(* CODESYS project machinemanage.library
   Title: MachineManage
   Version: 1.3.0.0
   Placeholder: MachineManage
   Company: Secote

Project tree, tasks and I/O mapping:
  libraries: Recipe Management, * (System); Tc2_DataExchange, * (Beckhoff Automation GmbH); Tc2_MC2, * (Beckhoff Automation GmbH); Tc2_MC2_Camming, * (Beckhoff Automation GmbH); Tc2_ModbusSrv, * (Beckhoff Automation GmbH); Tc2_Standard, * (Beckhoff Automation GmbH); Tc2_System, * (Beckhoff Automation GmbH); Tc2_TcpIp, * (Beckhoff Automation GmbH); Tc2_Utilities, * (Beckhoff Automation GmbH); Tc3_IotBase, * (Beckhoff Automation GmbH); Tc3_JsonXml, * (Beckhoff Automation GmbH); Tc3_MC2_AdvancedHoming, * (Beckhoff Automation GmbH); Tc3_PLCopen_OpcUa, * (Beckhoff Automation GmbH); VisuDialogs, * (System)
  Axis/
    DUTs/
      data type ST_Axis
      data type ST_AxisControl
      data type ST_AxisControlHome
      data type ST_AxisControlJog
      data type ST_AxisControlMove
      data type ST_AxisData
      data type ST_AxisInfo
      data type ST_AxisInput
      data type ST_AxisLock
      data type ST_AxisMode
      data type ST_AxisStatus
      data type ST_AxisTorque
    POUs/
      function block FB_Axis [ST]: A_ControlRest, A_Error, A_Home, A_Init, A_Jog, A_Memory, A_MoveAbsolute, A_MoveRelative, A_Power, A_Rest, A_Stop, A_Teach, M_GetAbsDone, M_GetRelDone, M_Home, M_Jog, M_MoveAbs, M_MoveRel
    VISUs/
      visualisation CtrlAxis
      visualisation CtrlAxisGroup
      text list TextHomeMode
  AxisCam/
    function block FB_AxisCam [ST]: A_Run, M_Semicircle
  Convert/
    function Data_TO_Data [ST]
  CycleTime/
    function block FB_CycleTime [ST]
    function block FB_CycleTime1 [ST]
  Cylinder/
    DUTs/
      data type ST_Cylinder
      data type ST_CylinderControl
      data type ST_CylinderData
      data type ST_CylinderInfo
      data type ST_CylinderInput
      data type ST_CylinderLock
      data type ST_CylinderOutput
      data type ST_CylinderStatus
    POUs/
      function block FB_Cylinder [ST]: A_ControlRest, A_Error, A_Home, A_Init, A_Memory, A_Off, A_Work, M_HomeRequest, M_OffRequest, M_WorkRequest
    VISUs/
      visualisation CtrlCylinder
      visualisation CtrlCylinderGroup
  Error/
    DUTs/
      data type E_ErrorCategory
      data type ST_Error
      data type ST_ErrorGroup
      data type ST_ErrorInfo
    POUs/
      function block FB_ErrorTag [ST]
      function block FB_ErrorTagStation [ST]
      function M_GetCategory [ST]
    VISUs/
      visualisation CtrlError
      visualisation CtrlError1
      visualisation CtrlErrorGroup
  File/
    DUTs/
      data type E_Directory
      data type ST_FileHandle
      data type ST_FileHandleData
      data type ST_FileHandleRead
      data type ST_FileHandleStatus
      data type ST_FilHandleControl
    POUs/
      function block FB_DirectoryHelper [ST]: A_Run
      function block FB_DirectoryHelper1 [ST]
      function block FB_FileHandle [ST]: A_Error, A_Read, A_Rest, A_Run, A_Status, A_Write
      function block FB_FileHelper [ST]
      function block FB_LogHelper [ST]: A_Run, A_Status
      function block FB_LogHelper_B [ST]: A_AddTail
      function block FB_LogHelper_E [ST]: A_Run, A_Status
      function block FB_LogHelper_E_B [ST]: A_AddTail
      function block FB_LogHelper1 [ST]: M_AddTail
  Hive/
    DUTs/
      data type E_HiveState
      data type ST_Hive
      data type ST_HiveAddress
      data type ST_HiveControl
      data type ST_HiveData
      data type ST_HiveInfo
      data type ST_HiveMachineData
    POUs/
      function block FB_Hive [ST]: A_Data, A_Init, A_Mode, A_State, A_Ton, M_Data, M_DateTime, M_Join0, M_ModeOff, M_ModeOn, M_State
      program P_Hive [ST]: M_Data, M_Error, M_GetData, M_Mode, M_State
  Http/
    DOTs/
      data type E_HttpRequestOrder
      data type ST_HttpClient
      data type ST_HttpClientControl
      data type ST_HttpClientData
      data type ST_HttpClientInfo
      data type ST_HttpClientStatus
    POUs/
      function block FB_HttpClient [ST]: A_Error, A_Init, A_Run, SendRequest
      function block FB_HttpClient1 [ST]: A_Run, SendRequest
    VISUs/
  ImagePool/
    Image/
      AlarmActive.png
      AlarmInactive.png
      AlarmInactive_gray.png
      auto_mode_80x80.png
      axis.png
      axis_black_80x80.png
      axis_gray_80x80.png
      axis_red_80x80.png
      background.png
      btn_off_switch.png
      btn_off_switch_silde.png
      btn_on_switch.png
      btn_on_switch_silde.png
      BtnData1.png
      BtnData2.png
      BtnFile1.png
      BtnFile2.png
      BtnHalt1.png
      BtnHalt2.png
      BtnHome1.png
      BtnHome2.png
      BtnInfo1.png
      BtnInfo2.png
      BtnLogin1.png
      BtnLogin2.png
      BtnOFF.png
      BtnON.png
      BtnPause1.png
      BtnPause2.png
      BtnSave1.png
      BtnSave2.png
      BtnSetting1.png
      BtnSetting2.png
      BtnStart1.png
      BtnStart2.png
      BtnVision1.png
      BtnVision2.png
      BtnVision3.png
      BtnVision4.png
      Button1.png
      Button10.png
      Button11.png
      Button13.png
      Button14.png
      Button15.png
      Button16.png
      Button17.png
      Button2.png
      Button3.png
      Button4.png
      Button5.png
      Button6.png
      Button7.png
      Button8.png
      Button9.png
      buzzer1.png
      buzzer2.png
      chinese.png
      cross-512.png
      Cylinder1.png
      English.png
      File.png
      Hindi.png
      ico_actuator_black.png
      ico_actuator_gray.png
      ico_actuator_red.png
      ico_analytic.png
      ico_analytic_100x100.png
      ico_analytic_off_100x100.png
      ico_apply.png
      ico_barcodeScanner.png
      ico_barcodeScanner_black.png
      ico_barcodeScanner_gray.png
      ico_barcodeScanner_red.png
      ico_calibrate.png
      ico_calibrate2.png
      ico_calibrate2_80x80.png
      ico_chart_bar.png
      ico_chart_half_pie.png
      ico_chart_line.png
      ico_chart_pie.png
      ico_clock_black.png
      ico_close.png
      ico_close_win.png
      ico_conveyor_big.png
      ico_conveyor_black.png
      ico_conveyor_gray.png
      ico_conveyor_red.png
      ico_diskdrive.png
      ico_folder.png
      ico_folder_.png
      ico_force_black_400X400.png
      ico_force_black_80X80.png
      ico_force_gray_80X80.png
      ico_force_red_80X80.png
      ico_HMI.png
      ico_info.png
      ico_io_300x300.png
      ico_max_win.png
      ico_menu_alarm.png
      ico_menu_backward.png
      ico_menu_camFolder.png
      ico_menu_clean.png
      ico_menu_excel.png
      ico_menu_forward.png
      ico_menu_home.png
      ico_menu_info.png
      ico_menu_options.png
      ico_menu_options_big.png
      ico_menu_pause.png
      ico_menu_play.png
      ico_menu_save.png
      ico_menu_stat.png
      ico_menu_step.png
      ico_menu_stop.png
      ico_menu_stop_black.png
      ico_menu_user.png
      ico_menu_user_logged_in.png
      ico_menu_vision.png
      ico_min_win.png
      ico_next.png
      ico_pneumatic_actuator.png
      ico_prev.png
      ico_robot_big.png
      ico_robot_black.png
      ico_robot_gray.png
      ico_robot_red.png
      ico_service.png
      ico_small_light_000.png
      ico_small_light_001.png
      ico_small_light_010.png
      ico_small_light_011.png
      ico_small_light_100.png
      ico_small_light_101.png
      ico_small_light_110.png
      ico_small_light_111.png
      ico_small_light_GGG.png
      ico_small_light_gray.png
      ico_small_light_green.png
      ico_small_light_red.png
      ico_stopper.png
      ico_tray.png
      ico_tray_black.png
      ico_tray_gray.png
      ico_tray_red.png
      ico_upload.png
      ico_usb.png
      ico_usb_small.png
      ico_vacuum_256x256.ico
      ico_vacuum_black_50x50.png
      ico_vacuum_cleaner_512x512.png
      ico_vacuum_cleaner_black_80x80.png
      ico_vacuum_cleaner_gray_80x80.png
      ico_vacuum_cleaner_red_80x80.png
      ico_vacuum_gray_50x50.png
      ico_vacuum_red_50x50.png
      ico_vacuumgauge_1200x1200.png
      ico_vacuumgauge_64x64.png
      ico_vacuumgauge_black_80x80.png
      ico_vacuumgauge_gray_80x80.png
      ico_vacuumgauge_red_80x80.png
      ico_version_history.png
      ico_vision_black.png
      ico_vision_gray.png
      ico_vision_red.png
      ico_wireless.png
      ico_wireless_51x40.png
      IO1.png
      IO2.png
      lamp.png
      lightbulb-default-80x80.png
      lightbulb-full-size.png
      lightbulb-off-80x80.png
      lightbulb-on-80x80.png
      Lock.jpg
      LUX.PNG
      manual_mode_80x80.png
      nav_first.png
      nav_last.png
      next.png
      NoImage.jpg
      phone.png
      phone1.png
      Pressure.png
      prev.png
      process.png
      right_arrow_128px_1205479_easyicon.net.ico
      right_arrow_128px_1205479_easyicon.net1.ico
      saveScreenshot.png
      service.png
      Setting.png
      Setting1.png
      Time.png
      Vietnamese.png
      warning.png
      zip_logs.png
    image pool ImagePool
  00000000-0000-0000-0000-000000000000|ImagePool\Image\AlarmActive.png
  00000000-0000-0000-0000-000000000000|ImagePool\Image\AlarmInactive.png
  00000000-0000-0000-0000-000000000000|ImagePool\Image\AlarmInactive_gray.png
  00000000-0000-0000-0000-000000000000|ImagePool\Image\auto_mode_80x80.png
  00000000-0000-0000-0000-000000000000|ImagePool\Image\axis.png
  00000000-0000-0000-0000-000000000000|ImagePool\Image\axis_black_80x80.png
  00000000-0000-0000-0000-000000000000|ImagePool\Image\axis_gray_80x80.png
  00000000-0000-0000-0000-000000000000|ImagePool\Image\axis_red_80x80.png
  00000000-0000-0000-0000-000000000000|ImagePool\Image\background.png
  00000000-0000-0000-0000-000000000000|ImagePool\Image\btn_off_switch.png
  00000000-0000-0000-0000-000000000000|ImagePool\Image\btn_off_switch_silde.png
  00000000-0000-0000-0000-000000000000|ImagePool\Image\btn_on_switch.png
  00000000-0000-0000-0000-000000000000|ImagePool\Image\btn_on_switch_silde.png
  00000000-0000-0000-0000-000000000000|ImagePool\Image\BtnData1.png
  00000000-0000-0000-0000-000000000000|ImagePool\Image\BtnData2.png
  00000000-0000-0000-0000-000000000000|ImagePool\Image\BtnFile1.png
  00000000-0000-0000-0000-000000000000|ImagePool\Image\BtnFile2.png
  00000000-0000-0000-0000-000000000000|ImagePool\Image\BtnHalt1.png
  00000000-0000-0000-0000-000000000000|ImagePool\Image\BtnHalt2.png
  00000000-0000-0000-0000-000000000000|ImagePool\Image\BtnHome1.png
  00000000-0000-0000-0000-000000000000|ImagePool\Image\BtnHome2.png
  00000000-0000-0000-0000-000000000000|ImagePool\Image\BtnInfo1.png
  00000000-0000-0000-0000-000000000000|ImagePool\Image\BtnInfo2.png
  00000000-0000-0000-0000-000000000000|ImagePool\Image\BtnLogin1.png
  00000000-0000-0000-0000-000000000000|ImagePool\Image\BtnLogin2.png
  00000000-0000-0000-0000-000000000000|ImagePool\Image\BtnOFF.png
  00000000-0000-0000-0000-000000000000|ImagePool\Image\BtnON.png
  00000000-0000-0000-0000-000000000000|ImagePool\Image\BtnPause1.png
  00000000-0000-0000-0000-000000000000|ImagePool\Image\BtnPause2.png
  00000000-0000-0000-0000-000000000000|ImagePool\Image\BtnSave1.png
  00000000-0000-0000-0000-000000000000|ImagePool\Image\BtnSave2.png
  00000000-0000-0000-0000-000000000000|ImagePool\Image\BtnSetting1.png
  00000000-0000-0000-0000-000000000000|ImagePool\Image\BtnSetting2.png
  00000000-0000-0000-0000-000000000000|ImagePool\Image\BtnStart1.png
  00000000-0000-0000-0000-000000000000|ImagePool\Image\BtnStart2.png
  00000000-0000-0000-0000-000000000000|ImagePool\Image\BtnVision1.png
  00000000-0000-0000-0000-000000000000|ImagePool\Image\BtnVision2.png
  00000000-0000-0000-0000-000000000000|ImagePool\Image\BtnVision3.png
  00000000-0000-0000-0000-000000000000|ImagePool\Image\BtnVision4.png
  00000000-0000-0000-0000-000000000000|ImagePool\Image\Button1.png
  00000000-0000-0000-0000-000000000000|ImagePool\Image\Button10.png
  00000000-0000-0000-0000-000000000000|ImagePool\Image\Button11.png
  00000000-0000-0000-0000-000000000000|ImagePool\Image\Button13.png
  00000000-0000-0000-0000-000000000000|ImagePool\Image\Button14.png
  00000000-0000-0000-0000-000000000000|ImagePool\Image\Button15.png
  00000000-0000-0000-0000-000000000000|ImagePool\Image\Button16.png
  00000000-0000-0000-0000-000000000000|ImagePool\Image\Button17.png
  00000000-0000-0000-0000-000000000000|ImagePool\Image\Button2.png
  00000000-0000-0000-0000-000000000000|ImagePool\Image\Button3.png
  00000000-0000-0000-0000-000000000000|ImagePool\Image\Button4.png
  00000000-0000-0000-0000-000000000000|ImagePool\Image\Button5.png
  00000000-0000-0000-0000-000000000000|ImagePool\Image\Button6.png
  00000000-0000-0000-0000-000000000000|ImagePool\Image\Button7.png
  00000000-0000-0000-0000-000000000000|ImagePool\Image\Button8.png
  00000000-0000-0000-0000-000000000000|ImagePool\Image\Button9.png
  00000000-0000-0000-0000-000000000000|ImagePool\Image\buzzer1.png
  00000000-0000-0000-0000-000000000000|ImagePool\Image\buzzer2.png
  00000000-0000-0000-0000-000000000000|ImagePool\Image\chinese.png
  00000000-0000-0000-0000-000000000000|ImagePool\Image\cross-512.png
  00000000-0000-0000-0000-000000000000|ImagePool\Image\Cylinder1.png
  00000000-0000-0000-0000-000000000000|ImagePool\Image\English.png
  00000000-0000-0000-0000-000000000000|ImagePool\Image\File.png
  00000000-0000-0000-0000-000000000000|ImagePool\Image\Hindi.png
  00000000-0000-0000-0000-000000000000|ImagePool\Image\ico_actuator_black.png
  00000000-0000-0000-0000-000000000000|ImagePool\Image\ico_actuator_gray.png
  00000000-0000-0000-0000-000000000000|ImagePool\Image\ico_actuator_red.png
  00000000-0000-0000-0000-000000000000|ImagePool\Image\ico_analytic.png
  00000000-0000-0000-0000-000000000000|ImagePool\Image\ico_analytic_100x100.png
  00000000-0000-0000-0000-000000000000|ImagePool\Image\ico_analytic_off_100x100.png
  00000000-0000-0000-0000-000000000000|ImagePool\Image\ico_apply.png
  00000000-0000-0000-0000-000000000000|ImagePool\Image\ico_barcodeScanner.png
  00000000-0000-0000-0000-000000000000|ImagePool\Image\ico_barcodeScanner_black.png
  00000000-0000-0000-0000-000000000000|ImagePool\Image\ico_barcodeScanner_gray.png
  00000000-0000-0000-0000-000000000000|ImagePool\Image\ico_barcodeScanner_red.png
  00000000-0000-0000-0000-000000000000|ImagePool\Image\ico_calibrate.png
  00000000-0000-0000-0000-000000000000|ImagePool\Image\ico_calibrate2.png
  00000000-0000-0000-0000-000000000000|ImagePool\Image\ico_calibrate2_80x80.png
  00000000-0000-0000-0000-000000000000|ImagePool\Image\ico_chart_bar.png
  00000000-0000-0000-0000-000000000000|ImagePool\Image\ico_chart_half_pie.png
  00000000-0000-0000-0000-000000000000|ImagePool\Image\ico_chart_line.png
  00000000-0000-0000-0000-000000000000|ImagePool\Image\ico_chart_pie.png
  00000000-0000-0000-0000-000000000000|ImagePool\Image\ico_clock_black.png
  00000000-0000-0000-0000-000000000000|ImagePool\Image\ico_close.png
  00000000-0000-0000-0000-000000000000|ImagePool\Image\ico_close_win.png
  00000000-0000-0000-0000-000000000000|ImagePool\Image\ico_conveyor_big.png
  00000000-0000-0000-0000-000000000000|ImagePool\Image\ico_conveyor_black.png
  00000000-0000-0000-0000-000000000000|ImagePool\Image\ico_conveyor_gray.png
  00000000-0000-0000-0000-000000000000|ImagePool\Image\ico_conveyor_red.png
  00000000-0000-0000-0000-000000000000|ImagePool\Image\ico_diskdrive.png
  00000000-0000-0000-0000-000000000000|ImagePool\Image\ico_folder.png
  00000000-0000-0000-0000-000000000000|ImagePool\Image\ico_folder_.png
  00000000-0000-0000-0000-000000000000|ImagePool\Image\ico_force_black_400X400.png
  00000000-0000-0000-0000-000000000000|ImagePool\Image\ico_force_black_80X80.png
  00000000-0000-0000-0000-000000000000|ImagePool\Image\ico_force_gray_80X80.png
  00000000-0000-0000-0000-000000000000|ImagePool\Image\ico_force_red_80X80.png
  00000000-0000-0000-0000-000000000000|ImagePool\Image\ico_HMI.png
  00000000-0000-0000-0000-000000000000|ImagePool\Image\ico_info.png
  00000000-0000-0000-0000-000000000000|ImagePool\Image\ico_io_300x300.png
  00000000-0000-0000-0000-000000000000|ImagePool\Image\ico_max_win.png
  00000000-0000-0000-0000-000000000000|ImagePool\Image\ico_menu_alarm.png
  00000000-0000-0000-0000-000000000000|ImagePool\Image\ico_menu_backward.png
  00000000-0000-0000-0000-000000000000|ImagePool\Image\ico_menu_camFolder.png
  00000000-0000-0000-0000-000000000000|ImagePool\Image\ico_menu_clean.png
  00000000-0000-0000-0000-000000000000|ImagePool\Image\ico_menu_excel.png
  00000000-0000-0000-0000-000000000000|ImagePool\Image\ico_menu_forward.png
  00000000-0000-0000-0000-000000000000|ImagePool\Image\ico_menu_home.png
  00000000-0000-0000-0000-000000000000|ImagePool\Image\ico_menu_info.png
  00000000-0000-0000-0000-000000000000|ImagePool\Image\ico_menu_options.png
  00000000-0000-0000-0000-000000000000|ImagePool\Image\ico_menu_options_big.png
  00000000-0000-0000-0000-000000000000|ImagePool\Image\ico_menu_pause.png
  00000000-0000-0000-0000-000000000000|ImagePool\Image\ico_menu_play.png
  00000000-0000-0000-0000-000000000000|ImagePool\Image\ico_menu_save.png
  00000000-0000-0000-0000-000000000000|ImagePool\Image\ico_menu_stat.png
  00000000-0000-0000-0000-000000000000|ImagePool\Image\ico_menu_step.png
  00000000-0000-0000-0000-000000000000|ImagePool\Image\ico_menu_stop.png
  00000000-0000-0000-0000-000000000000|ImagePool\Image\ico_menu_stop_black.png
  00000000-0000-0000-0000-000000000000|ImagePool\Image\ico_menu_user.png
  00000000-0000-0000-0000-000000000000|ImagePool\Image\ico_menu_user_logged_in.png
  00000000-0000-0000-0000-000000000000|ImagePool\Image\ico_menu_vision.png
  00000000-0000-0000-0000-000000000000|ImagePool\Image\ico_min_win.png
  00000000-0000-0000-0000-000000000000|ImagePool\Image\ico_next.png
  00000000-0000-0000-0000-000000000000|ImagePool\Image\ico_pneumatic_actuator.png
  00000000-0000-0000-0000-000000000000|ImagePool\Image\ico_prev.png
  00000000-0000-0000-0000-000000000000|ImagePool\Image\ico_robot_big.png
  00000000-0000-0000-0000-000000000000|ImagePool\Image\ico_robot_black.png
  00000000-0000-0000-0000-000000000000|ImagePool\Image\ico_robot_gray.png
  00000000-0000-0000-0000-000000000000|ImagePool\Image\ico_robot_red.png
  00000000-0000-0000-0000-000000000000|ImagePool\Image\ico_service.png
  00000000-0000-0000-0000-000000000000|ImagePool\Image\ico_small_light_000.png
  00000000-0000-0000-0000-000000000000|ImagePool\Image\ico_small_light_001.png
  00000000-0000-0000-0000-000000000000|ImagePool\Image\ico_small_light_010.png
  00000000-0000-0000-0000-000000000000|ImagePool\Image\ico_small_light_011.png
  00000000-0000-0000-0000-000000000000|ImagePool\Image\ico_small_light_100.png
  00000000-0000-0000-0000-000000000000|ImagePool\Image\ico_small_light_101.png
  00000000-0000-0000-0000-000000000000|ImagePool\Image\ico_small_light_110.png
  00000000-0000-0000-0000-000000000000|ImagePool\Image\ico_small_light_111.png
  00000000-0000-0000-0000-000000000000|ImagePool\Image\ico_small_light_GGG.png
  00000000-0000-0000-0000-000000000000|ImagePool\Image\ico_small_light_gray.png
  00000000-0000-0000-0000-000000000000|ImagePool\Image\ico_small_light_green.png
  00000000-0000-0000-0000-000000000000|ImagePool\Image\ico_small_light_red.png
  00000000-0000-0000-0000-000000000000|ImagePool\Image\ico_stopper.png
  00000000-0000-0000-0000-000000000000|ImagePool\Image\ico_tray.png
  00000000-0000-0000-0000-000000000000|ImagePool\Image\ico_tray_black.png
  00000000-0000-0000-0000-000000000000|ImagePool\Image\ico_tray_gray.png
  00000000-0000-0000-0000-000000000000|ImagePool\Image\ico_tray_red.png
  00000000-0000-0000-0000-000000000000|ImagePool\Image\ico_upload.png
  00000000-0000-0000-0000-000000000000|ImagePool\Image\ico_usb.png
  00000000-0000-0000-0000-000000000000|ImagePool\Image\ico_usb_small.png
  00000000-0000-0000-0000-000000000000|ImagePool\Image\ico_vacuum_256x256.ico
  00000000-0000-0000-0000-000000000000|ImagePool\Image\ico_vacuum_black_50x50.png
  00000000-0000-0000-0000-000000000000|ImagePool\Image\ico_vacuum_cleaner_512x512.png
  00000000-0000-0000-0000-000000000000|ImagePool\Image\ico_vacuum_cleaner_black_80x80.png
  00000000-0000-0000-0000-000000000000|ImagePool\Image\ico_vacuum_cleaner_gray_80x80.png
  00000000-0000-0000-0000-000000000000|ImagePool\Image\ico_vacuum_cleaner_red_80x80.png
  00000000-0000-0000-0000-000000000000|ImagePool\Image\ico_vacuum_gray_50x50.png
  00000000-0000-0000-0000-000000000000|ImagePool\Image\ico_vacuum_red_50x50.png
  00000000-0000-0000-0000-000000000000|ImagePool\Image\ico_vacuumgauge_1200x1200.png
  00000000-0000-0000-0000-000000000000|ImagePool\Image\ico_vacuumgauge_64x64.png
  00000000-0000-0000-0000-000000000000|ImagePool\Image\ico_vacuumgauge_black_80x80.png
  00000000-0000-0000-0000-000000000000|ImagePool\Image\ico_vacuumgauge_gray_80x80.png
  00000000-0000-0000-0000-000000000000|ImagePool\Image\ico_vacuumgauge_red_80x80.png
  00000000-0000-0000-0000-000000000000|ImagePool\Image\ico_version_history.png
  00000000-0000-0000-0000-000000000000|ImagePool\Image\ico_vision_black.png
  00000000-0000-0000-0000-000000000000|ImagePool\Image\ico_vision_gray.png
  00000000-0000-0000-0000-000000000000|ImagePool\Image\ico_vision_red.png
  00000000-0000-0000-0000-000000000000|ImagePool\Image\ico_wireless.png
  00000000-0000-0000-0000-000000000000|ImagePool\Image\ico_wireless_51x40.png
  00000000-0000-0000-0000-000000000000|ImagePool\Image\IO1.png
  00000000-0000-0000-0000-000000000000|ImagePool\Image\IO2.png
  00000000-0000-0000-0000-000000000000|ImagePool\Image\lamp.png
  00000000-0000-0000-0000-000000000000|ImagePool\Image\lightbulb-default-80x80.png
  00000000-0000-0000-0000-000000000000|ImagePool\Image\lightbulb-full-size.png
  00000000-0000-0000-0000-000000000000|ImagePool\Image\lightbulb-off-80x80.png
  00000000-0000-0000-0000-000000000000|ImagePool\Image\lightbulb-on-80x80.png
  00000000-0000-0000-0000-000000000000|ImagePool\Image\Lock.jpg
  00000000-0000-0000-0000-000000000000|ImagePool\Image\LUX.PNG
  00000000-0000-0000-0000-000000000000|ImagePool\Image\manual_mode_80x80.png
  00000000-0000-0000-0000-000000000000|ImagePool\Image\nav_first.png
  00000000-0000-0000-0000-000000000000|ImagePool\Image\nav_last.png
  00000000-0000-0000-0000-000000000000|ImagePool\Image\next.png
  00000000-0000-0000-0000-000000000000|ImagePool\Image\NoImage.jpg
  00000000-0000-0000-0000-000000000000|ImagePool\Image\phone.png
  00000000-0000-0000-0000-000000000000|ImagePool\Image\phone1.png
  00000000-0000-0000-0000-000000000000|ImagePool\Image\Pressure.png
  00000000-0000-0000-0000-000000000000|ImagePool\Image\prev.png
  00000000-0000-0000-0000-000000000000|ImagePool\Image\process.png
  00000000-0000-0000-0000-000000000000|ImagePool\Image\right_arrow_128px_1205479_easyicon.net.ico
  00000000-0000-0000-0000-000000000000|ImagePool\Image\right_arrow_128px_1205479_easyicon.net1.ico
  00000000-0000-0000-0000-000000000000|ImagePool\Image\saveScreenshot.png
  00000000-0000-0000-0000-000000000000|ImagePool\Image\service.png
  00000000-0000-0000-0000-000000000000|ImagePool\Image\Setting.png
  00000000-0000-0000-0000-000000000000|ImagePool\Image\Setting1.png
  00000000-0000-0000-0000-000000000000|ImagePool\Image\Time.png
  00000000-0000-0000-0000-000000000000|ImagePool\Image\Vietnamese.png
  00000000-0000-0000-0000-000000000000|ImagePool\Image\warning.png
  00000000-0000-0000-0000-000000000000|ImagePool\Image\zip_logs.png
  IO/
    visualisation CtrlInput
    visualisation CtrlOutput
    text list InputText
    text list OutputText
  Json/
    POUs/
      function block FB_JsonObjV5 [ST]: A_FileJsonObj, M_AddKeyValue, M_GetJsonStr, M_GetKeyValue, M_JsonStrToObj, M_ObjToJsonStr, M_ResetObj
  Matrix2D/
    function block FB_Matrix2D [ST]: M_Index_S, M_Index_Z, M_XY
    data type ST_Matrix2DCoordinate
  ModbusTcp/
    data type E_ModbusClientTcpCmd
    function block FB_ModbusTcpClient [ST]: A_Run
  OpcUa/
    DOTs/
      data type E_OpcUaClientCmd
    POUS/
      function block FB_OpcUaClient [ST]: A_Run
  Recipe/
    POUs/
      program P_Recipe [ST]
    VISUs/
      visualisation CtrlRecipe
  Regex/
    function F_FIND [ST]
    function F_Join [ST]
    function F_Join_L [ST]
    function F_Join_L1 [ST]
    function F_LEN [ST]
    function F_MID [ST]
    function F_Split [ST]
    function F_WString_TO_String_UTF8 [ST]
    function M_Join0 [ST]
  System/
    DUTs/
      data type E_Language
      data type ST_Status
      data type ST_System
      data type ST_SystemDate
      data type ST_SystemInput
      data type ST_SystemLog
      data type ST_SystemMode
      data type ST_SystemOutput
      data type ST_SystemStation
      data type ST_SystemStationHistory
      data type ST_TriggerMode
    POUs/
      function block FB_AutoAgain [ST]
      function block FB_Beacon [ST]
      function block FB_Bool [ST]: M_F_TRIG, M_R_TRIG, M_TON
      function block FB_Button [ST]
      function block FB_Memory [ST]
      function block FB_Memory1 [ST]
      function block FB_MemoryLag [ST]
      function block FB_Pulse [ST]
      function block FB_System [ST]: A_Log, A_ModeAlarm, A_ModeAuto, A_ModeAutoRunning, A_ModeBreakpoint, A_ModeDevice, A_ModeEtop, A_ModeHomeDone, A_ModeHoming, A_ModeInit, A_ModeManual, A_ModeMemory, A_ModeNone, A_ModePause, A_ModeSetting, A_ModeStop, A_NowMode, A_StepAlternate, A_SystemDate
    VISUs/
      visualisation CtrlAxisCylinder
      visualisation CtrlBtnBox
      visualisation CtrlBtnLogin
      visualisation CtrlFormColse
      visualisation CtrlHomeGroup
      visualisation CtrlLanguage
      visualisation CtrlMode
      visualisation CtrlPageSwitch
      visualisation CtrlStation
  TcpIp/
    DUTs/
      data type E_TcpIpClientCmd
      data type ST_TcpIpClient
      data type ST_TcpIpClientControl
      data type ST_TcpIpClientInfo
      data type ST_TcpIpClientStatus
      data type ST_TcpIpData
    POUs/
      function block FB_TcpIpClient [ST]: A_Close, A_Connect, A_ControlReset, A_Error, A_Init, A_Receive, A_Send, A_Status
      function block FB_TcpIpClient1 [ST]: A_Run
    VISUs/
      visualisation CtrlTcpIpClient
  Version/
    global variables Global_Version
  Windows/
    function block FB_WindowsCmd [ST]: A_Run
    function block FB_WindowsCmdAsync [ST]: A_Run
  Yield/
    DUTs/
      data type ST_Yield
      data type ST_YieldControl
      data type ST_YieldData
    POUs/
      function block FB_Yield [ST]
    VISUs/
      visualisation CtrlYield
  text list GlobalTextList
  global variables GVL
  global variables GVL_Data_P
  global variables GVL_P
  program P_Machine [ST]
*)

// Axis/DUTs/ST_Axis
TYPE ST_Axis :
STRUCT
	ID:									BYTE;
	stInput:							ST_AxisInput;// 轴IO接口
	stLock:								ST_AxisLock;// 轴动作安全锁
	stStatus:							ST_AxisStatus;// 轴状态
	stControl:							ST_AxisControl;// 轴控制
	Axis_REF:							AXIS_REF;// 虚拟轴接口
	arrInfo:							ARRAY[0..E_Language.MaxCount] OF ST_AxisInfo;
	
	{attribute'hide'}
	sName:								WSTRING;// 当前语言名称(只读)
END_STRUCT
END_TYPE

// Axis/DUTs/ST_AxisControl
TYPE ST_AxisControl :
STRUCT
	stJog:					ST_AxisControlJog;// 点动控制
	stStop:					ST_TriggerMode;// 轴停止
	stHome:					ST_TriggerMode;// 回零
	stReset:				ST_TriggerMode;// 轴整体复位
	stMovePosition:			ST_AxisControlMove;// 定位(包含绝对定位和相对定位)	
	stClosePower:			ST_TriggerMode;// 伺服断使能(目前只有手动控制 才可以断伺服使能)
	stTeach:				ST_TriggerMode;// 示教
	stMoveMemory:			ST_TriggerMode;// 至记忆位
END_STRUCT
END_TYPE

// Axis/DUTs/ST_AxisControlHome
TYPE ST_AxisControlHome :
STRUCT
	iDirection:						INT;// -1:反向回零;0:直接回零;1:先到正向回零
	stStartHome:					ST_TriggerMode;// 启动回零
END_STRUCT
END_TYPE

// Axis/DUTs/ST_AxisControlJog
TYPE ST_AxisControlJog :
STRUCT
	stPositive:					ST_TriggerMode;// 点动正转
	stNegative:					ST_TriggerMode;// 点动反转
END_STRUCT
END_TYPE

// Axis/DUTs/ST_AxisControlMove
TYPE ST_AxisControlMove :
STRUCT
	iIndex:						UINT;// 定位索引
	stStartAbs:					ST_TriggerMode;// 开始绝对定位
	stStartRel:					ST_TriggerMode;// 开始相对定位
END_STRUCT
END_TYPE

// Axis/DUTs/ST_AxisData
TYPE ST_AxisData :
STRUCT
	fJogVelocity:					LREAL;// 点动速度
	fJogAccelerated:				LREAL:=5000;// 点动加速度
	fJogDeceleration:				LREAL:=5000;// 点动减速度
	arrMoveAccelerated:				ARRAY [0..20]OF LREAL:=[5000,5000,5000,5000,5000,5000,5000,5000,5000,5000,5000,5000,5000,5000,5000,5000,5000,5000,5000,5000,5000];// 定位加速度
	arrMoveDeceleration:			ARRAY [0..20]OF LREAL:=[5000,5000,5000,5000,5000,5000,5000,5000,5000,5000,5000,5000,5000,5000,5000,5000,5000,5000,5000,5000,5000];// 定位减速度
	arrMovePosition:				ARRAY[0..20]OF LREAL;// 定位位置
	arrMoveVelocity:				ARRAY[0..20]OF LREAL;// 定位速度
	stTorque:						ST_AxisTorque;// 力矩
	stMode:							ST_AxisMode;// 模式
	iSetHomeVelocity:				LREAL:=0.05;// 速度回零及扭矩回零监控最小速度
	iSetMoveFluctuation:			LREAL:=0.01;// 定位允许误差 (正实数);
	
	fMemoryPosition:				LREAL;// 轴记忆位置
END_STRUCT
END_TYPE

// Axis/DUTs/ST_AxisInfo
TYPE ST_AxisInfo :
STRUCT
	sName:						WSTRING;// 轴名称
	sFbErrorInfo:				WSTRING;// 功能块错误提示
	sNegativeInfo:				WSTRING;// 负极限错误提示
	sPositiveInfo:				WSTRING;// 正极限错误提示
	sHomeInfo:					WSTRING;// 回零超时错误提示
	sMemoryPos:					WSTRING;// 记忆位置
END_STRUCT
END_TYPE

// Axis/DUTs/ST_AxisInput
TYPE ST_AxisInput :
STRUCT
	bPositive:							BOOL;// 正极限
	bNegative:							BOOL;// 负极限
END_STRUCT
END_TYPE

// Axis/DUTs/ST_AxisLock
TYPE ST_AxisLock :
STRUCT
	bHome:					BOOL;// 回零安全锁
	arrMovePosition:		ARRAY[0..20]OF BOOL;// 定位位置锁
	bJogPositive:			BOOL;// 点动正转锁
	bJogNegative:			BOOL;// 点动反转锁	
	bAll:					BOOL;// 总状态锁
	bShield:				BOOL;// 屏蔽整个功能块
	bMoveAbsAll:			BOOL;// 绝对定位 位置总锁
	bMoveRelAll:			BOOL;// 相对定位 位置总锁	
END_STRUCT
END_TYPE

// Axis/DUTs/ST_AxisMode
TYPE ST_AxisMode :
STRUCT
	iHomeMode:						INT;// 回零模式(0:采集原点回零;1:力矩反馈回零;2:定义当前位置为原点)
END_STRUCT
END_TYPE

// Axis/DUTs/ST_AxisStatus
TYPE ST_AxisStatus :
STRUCT
	bError:				BOOL;// 错误
	iErrorID:			UDINT;// 错误代码
	bPowered:			BOOL;// 上电完成
	bMoving:			BOOL;// 运动中
	bHoming:			BOOL;// 回零中
	bHomeDone:			BOOL;// 回零完成
	bMoveAbsDone:		BOOL;// 绝对定位完成
	bMoveRelDone:		BOOL;// 相对定位完成
	bErrorFB:			BOOL;// 功能块错误
	bErrorNegative:		BOOL;// 碰负极限
	bErrorPositive:		BOOL;// 碰正极限
	bErrorHome:			BOOL;// 回零超时
	bMemoryPos:			BOOL;// 记忆位置
END_STRUCT
END_TYPE

// Axis/DUTs/ST_AxisTorque
TYPE ST_AxisTorque :
STRUCT
	iGetTorque:						INT;// 当前力矩
	iSetTorque:						INT;// 设置力矩
END_STRUCT
END_TYPE

// Cylinder/DUTs/ST_Cylinder
TYPE ST_Cylinder :
STRUCT
	ID:					BYTE;
	stInput:			ST_CylinderInput;// 输入
	stOutput:			ST_CylinderOutput;// 输出
	stControl:			ST_CylinderControl;// 控制
	stLock:				ST_CylinderLock;// 安全锁
	stStatus:			ST_CylinderStatus;// 状态
	arrInfo:			ARRAY[0..E_Language.MaxCount] OF ST_CylinderInfo;// 提示信息
	{attribute'hide'}
	sName:				WSTRING;// 当前语言名称(只读)
END_STRUCT
END_TYPE

// Cylinder/DUTs/ST_CylinderControl
TYPE ST_CylinderControl :
STRUCT
	stWorkRequest:		ST_TriggerMode;// 动作请求
	stHomeRequest:		ST_TriggerMode;// 复位请求
	stOffRequest:		ST_TriggerMode;// 释放请求
END_STRUCT
END_TYPE

// Cylinder/DUTs/ST_CylinderData
TYPE ST_CylinderData :
STRUCT
	iAlarmTime:			UDINT:=3000;// 报警延迟ms
	iHomeRequestTime:	UDINT;// 动作延迟
	iWorkRequestTime:	UDINT;// 动作延迟
	iOffRequestTime:	UDINT;// 动作延迟
	iHomeDone:			UDINT;// 到位延迟
	iWorkDone:			UDINT;// 到位延迟
	iOffDone:			UDINT;// 到位延迟
END_STRUCT
END_TYPE

// Cylinder/DUTs/ST_CylinderInfo
TYPE ST_CylinderInfo :
STRUCT
	sName:				WSTRING;// 名称
	sHomeError:			WSTRING;// 初始位提示报警
	sWorkError:			WSTRING;// 工作位提示报警
	sWorkHomeError:		WSTRING;// 工作位 初始位同时有信号
	sMemoryHome:		WSTRING;// 初始位记忆提示信息
	sMemoryWork:		WSTRING;// 工作位记忆提示信息
END_STRUCT
END_TYPE

// Cylinder/DUTs/ST_CylinderInput
TYPE ST_CylinderInput :
STRUCT
	bWork:				  BOOL;// 工作位
	bHome:				  BOOL;// 初始位
END_STRUCT
END_TYPE

// Cylinder/DUTs/ST_CylinderLock
TYPE ST_CylinderLock :
STRUCT
	bWork:					BOOL;// 工作锁
	bHome:					BOOL;// 初始锁
	bOff:					BOOL;// 释放锁
	bAll:					BOOL;// 总状态锁
	bShield:				BOOL;// 屏蔽整个功能块
END_STRUCT
END_TYPE

// Cylinder/DUTs/ST_CylinderOutput
TYPE ST_CylinderOutput :
STRUCT
	bWork:			BOOL;// 工作位
	bHome:			BOOL;// 初始位
END_STRUCT
END_TYPE

// Cylinder/DUTs/ST_CylinderStatus
TYPE ST_CylinderStatus :
STRUCT
	bErrorHome:			BOOL;// 回初始位错误
	bErrorWork:			BOOL;// 回工作位错误
	bErrorTogether:		BOOL;// 传感器同时有信号
	bMemoryHome:		BOOL;// 初始位和记忆状态不符合
	bMemoryWork:		BOOL;// 工作位和记忆状态不符合
	
	bHomeDone:			BOOL;// 初始位到位延迟
	bWorkDone:			BOOL;// 工作位到位延迟
	bOffDone:			BOOL;// 中间位到位延迟
END_STRUCT
END_TYPE

// Error/DUTs/E_ErrorCategory
{attribute 'qualified_only'}
{attribute 'strict'}
TYPE E_ErrorCategory :
(
	Safety:=1,// 安全类
	Cylinder,// 气缸类
	Axis,// 轴类
	Station,// 工站流程类
	TCP_IP,// TCP通信类
	File,// 文件操作
	Http,// Http通信类
	Other// 其他
);
END_TYPE

// Error/DUTs/ST_Error
TYPE ST_Error :
STRUCT
	bSaveLog:		BOOL;
	bSaveErrorList:	BOOL;
	sFileLogPath:	STRING;// Log保存文件夹路径
	eLanguage:		E_Language:=E_Language.Chinese;// Log保存的语言
	eSaveListLanguage:	E_Language:=E_Language.English;// 保存成ErrorList的语言
	stNow:			ST_ErrorGroup;// 当前报警集合
	stHistory:		ST_ErrorGroup;// 历史报警集合
END_STRUCT
END_TYPE

// Error/DUTs/ST_ErrorGroup
TYPE ST_ErrorGroup :
STRUCT
	iCount:			INT:=20;
	arrInfo:		ARRAY[0..20] OF ST_ErrorInfo;
END_STRUCT
END_TYPE

// Error/DUTs/ST_ErrorInfo
TYPE ST_ErrorInfo :
STRUCT
	bStatus:				BOOL;// 报警状态
	sSystemDate:			STRING;// 报警时间
	sLevel:					STRING;// 报警等级
	sPosition:				WSTRING;// 错误发生位置
	iErrorCode:				DWORD;// 报警代码
	arrMessage:				ARRAY[0..E_Language.MaxCount] OF WSTRING;// 报警信息
END_STRUCT
END_TYPE

// File/DUTs/E_Directory
{attribute 'qualified_only'}
{attribute 'strict'}
TYPE E_Directory :
(
	Create,
	Delete
);
END_TYPE

// File/DUTs/ST_FileHandle
TYPE ST_FileHandle :
STRUCT
	ID:								BYTE;
	sName:							WSTRING;// 名称
	stStatus:						ST_FileHandleStatus;// 状态
	stControl:						ST_FilHandleControl;// 控制
	stReadBuffer:					ST_FileHandleRead;
	sWriteBuffer:					STRING(255);
END_STRUCT
END_TYPE

// File/DUTs/ST_FileHandleData
TYPE ST_FileHandleData :
STRUCT
	sFilePath:					STRING;// 文件路径
END_STRUCT
END_TYPE

// File/DUTs/ST_FileHandleRead
TYPE ST_FileHandleRead :
STRUCT
	iCount:					INT:=99;
	arrBuffer:				ARRAY[0..99] OF STRING;
	iLength:				INT;//  读取后实际 缓存区长度
END_STRUCT
END_TYPE

// File/DUTs/ST_FileHandleStatus
TYPE ST_FileHandleStatus :
STRUCT
	bDone:					BOOL;// 完成
	bBusy:					BOOL;// 进行中
	bError:					BOOL;// 错误
	iErrorID:				UDINT;// 错误代码
	bErrorOpen:				BOOL;// 文件打开错误
	bErrorGet:				BOOL;// 文件读取错误
	bErrorWrite:			BOOL;// 文件写入错误
	bErrorClose:			BOOL;// 文件关闭错误	
END_STRUCT
END_TYPE

// File/DUTs/ST_FilHandleControl
TYPE ST_FilHandleControl :
STRUCT
	stRead:						ST_TriggerMode;// 读取
	stWrite:					ST_TriggerMode;// 写入
END_STRUCT
END_TYPE

// Hive/DUTs/E_HiveState
{attribute 'qualified_only'}
{attribute 'strict'}
TYPE E_HiveState :
(	
	None:=0,
	Running,// 运行中
	Idle,// 空闲状态
	Engineering,// 管理模式
	PlannedDown,// 计划停机
	UnplannedDown// 非计划停机
);
END_TYPE

// Hive/DUTs/ST_Hive
TYPE ST_Hive :
STRUCT
	stControl:			ST_HiveControl;// 控制
	eState:				E_HiveState;// 当前设备状态 只读
	stSendDataState:	ST_Status;
END_STRUCT
END_TYPE

// Hive/DUTs/ST_HiveAddress
TYPE ST_HiveAddress :
STRUCT
	sIP:					STRING;// 服务器地址
	iPort:					UINT;// 服务器端口号
	sUri:					STRING;// 网址
END_STRUCT
END_TYPE

// Hive/DUTs/ST_HiveControl
TYPE ST_HiveControl :
STRUCT
	bStateEnable:		BOOL;// 启用状态发送
	bModeEnable:		BOOL;// 启用模式发送
	bDataEnable:		BOOL;// 启用数据发送
	bPlannedDown:		BOOL;// 计划停机
	bSendData:			BOOL;// 发送数据
	bModeLogin:			BOOL;// 模式登录(true:登录;false:登录退出);需保持信号
	stMachineData:		ST_HiveMachineData;
	sSession_token:		STRING;// Mode登录令牌
	arrActivity:		POINTER TO STRING;
	iActivityCount:		INT;// arrActivity元素数量
END_STRUCT
END_TYPE

// Hive/DUTs/ST_HiveData
TYPE ST_HiveData :
STRUCT
	stStateAddress:				ST_HiveAddress;
	stModeAddressOn:			ST_HiveAddress;
	stModeAddressOff:			ST_HiveAddress;
	stDataAddress:				ST_HiveAddress;
	iTimeOut:					UINT:=3000;// 通信超时(ms)
	eLanguage:					E_Language:=E_Language.English;// 上传的语言
END_STRUCT
END_TYPE

// Hive/DUTs/ST_HiveInfo
TYPE ST_HiveInfo :
STRUCT
	sName:					WSTRING;
END_STRUCT
END_TYPE

// Hive/DUTs/ST_HiveMachineData
TYPE ST_HiveMachineData :
STRUCT
	sUnit_sn:		STRING;
	sCarrier_sn:	STRING;
	sWip_serials:	STRING;
	bPass:			BOOL;
	sInput_time:	STRING;
	sOutput_time:	STRING;
	arrDataName:	POINTER TO STRING;
	arrDataValue:	POINTER TO STRING;
	iDataCount:		INT;
END_STRUCT
END_TYPE

// Http/DOTs/E_HttpRequestOrder
{attribute 'qualified_only'}
{attribute 'strict'}
TYPE E_HttpRequestOrder :
(
	None :=0,
	GET,
	POST
);
END_TYPE

// Http/DOTs/ST_HttpClient
TYPE ST_HttpClient :
STRUCT
	ID:								BYTE;
	sName:							WSTRING;// 当前语言名称(只读)
	stControl:						ST_HttpClientControl;// 控制
	stStatus:						ST_HttpClientStatus;// 状态
	arrInfo:						ARRAY[0..E_Language.MaxCount] OF ST_HttpClientInfo;
END_STRUCT
END_TYPE

// Http/DOTs/ST_HttpClientControl
TYPE ST_HttpClientControl :
STRUCT
	eRequest:					E_HttpRequestOrder;// 客户端请求服务器命令
	sRequestData:				STRING(5000);// 客户端请求服务器数据
	sResponseData:				STRING(5000);// 服务器响应数据
END_STRUCT
END_TYPE

// Http/DOTs/ST_HttpClientData
TYPE ST_HttpClientData :
STRUCT
	sIP:					STRING;// 服务器地址
	iPort:					UINT;// 服务器端口号
	sUri:					STRING;// 网址
	iTimeOut:				UINT:=6000;// 通信超时(ms)
END_STRUCT
END_TYPE

// Http/DOTs/ST_HttpClientInfo
TYPE ST_HttpClientInfo :
STRUCT
	sName:					WSTRING;
	sError:					WSTRING;// 状态错误
	sErrorTimeOut:			WSTRING;// 超时错误
END_STRUCT
END_TYPE

// Http/DOTs/ST_HttpClientStatus
TYPE ST_HttpClientStatus :
STRUCT
	bBusy:				BOOL;
	bDone:				BOOL;
	bError:				BOOL;
	iErrorID:			INT;
	bErrorTimeOut:		BOOL;// 超时错误
END_STRUCT
END_TYPE

// Matrix2D/ST_Matrix2DCoordinate
TYPE ST_Matrix2DCoordinate :
STRUCT
	X:					LREAL;
	Y:					LREAL;
END_STRUCT
END_TYPE

// ModbusTcp/E_ModbusClientTcpCmd
{attribute 'qualified_only'}
{attribute 'strict'}
TYPE E_ModbusClientTcpCmd :
(
	None := 0,
	ReadCoils,// 读取多个线圈
	ReadRegs,// 读取多个寄存器
	WriteRegs,// 写入多个寄存器
	WriteCoils,// 写入多个线圈
	Reset// 复位
	
);
END_TYPE

// OpcUa/DOTs/E_OpcUaClientCmd
{attribute 'qualified_only'}
{attribute 'strict'}
TYPE E_OpcUaClientCmd :
(
	None:=0,
	Read:=1,
	Write:=2,
	Connect:=100,
	Disconnect:=101,
	Reset
);
END_TYPE

// System/DUTs/E_Language
{attribute 'qualified_only'}
{attribute 'strict'}
TYPE E_Language :
(
	Chinese:=0,// 简体中文
	English,// 英语
	Vietnamese,// 越南语
	Hindi,// 印度语
	Standby1,// 备用1
	Standby2,// 备用2
	MaxCount
);
END_TYPE

// System/DUTs/ST_Status
TYPE ST_Status :
STRUCT
	bBusy:				BOOL;
	bDone:				BOOL;
	bError:				BOOL;
END_STRUCT
END_TYPE

// System/DUTs/ST_System
TYPE ST_System :
STRUCT
	stInput:				ST_SystemInput;// 输入
	stOutput:				ST_SystemOutput;// 输出
	stMode:					ST_SystemMode;// 设备状态			
	stSystemDate:			ST_SystemDate;// 系统时间
	stLogConfig:			ST_SystemLog;// Log配置
	
	{attribute'hide'}
	iSafetyLevel:			INT:=5;// 安全等级
	iPageNow:				INT;
END_STRUCT
END_TYPE

// System/DUTs/ST_SystemDate
TYPE ST_SystemDate :
STRUCT
	iYear:						INT;// 年
	iMonth:						INT;// 月
	iDay:						INT;// 日
	iHour:						INT;// 小时
	iMinute:					INT;// 分钟
	iSecond:					INT;// 秒
	iMilliseconds:				INT;// 毫秒
	sNow:						STRING;// 当前完整时间
	sDateDay:					STRING;// 时间到天(yy/MM/dd)
END_STRUCT
END_TYPE

// System/DUTs/ST_SystemInput
TYPE ST_SystemInput :
STRUCT
	bAuto:				BOOL;// 自动
	bManual:			BOOL;// 手动
	bEStop:				BOOL;// 急停
	bStart:				BOOL;// 启动
	bPause:				BOOL;// 暂停
	bStop:				BOOL;// 停止
	bReset:				BOOL;// 复位
	bResetAlarm:		BOOL;// 复位报警
	bQuiet:				BOOL;// 静音
	bSetting:			BOOL;// 设置
	bInit:				BOOL;// 初始化
END_STRUCT
END_TYPE

// System/DUTs/ST_SystemLog
TYPE ST_SystemLog :
STRUCT
	sFilePath:			STRING;// 文件夹路径
	bExecute:			BOOL;// 执行	
	eLanguage:			E_Language:=E_Language.Chinese;// Log保存语言	
END_STRUCT
END_TYPE

// System/DUTs/ST_SystemMode
TYPE ST_SystemMode :
STRUCT
	bAuto:					BOOL;// 自动状态
	bPause:					BOOL;// 暂停
	bAutoRunning:			BOOL;// 自动运行
	bHoming:				BOOL;// 初始中
	bHomeDone:				BOOL;// 初始化完成
	bManual:				BOOL;// 手动状态
	arrAlarm:				ARRAY[1..5]OF BOOL;// 报警状态
	arrAlarmStation:		ARRAY[0..100] OF BOOL;// 当工站报警状态
	bStop:					BOOL;// 停止状态
	bEStop:					BOOL;// 急停状态
	stDeviceEnable: 		ST_TriggerMode;// 允许执行元件 动作
	stDeviceRest:			ST_TriggerMode;// 执行元件 控制复位
	bSetting:				BOOL;// 设置模式
	iMemory:				INT;// 记忆(用于记录 轴或气缸等执行元件 在自动状态下 人工干预次数)
	bAlarming:				BOOL;// 报警中
	sNowMode:				STRING;// 设备当前模式
	bNone:					BOOL;// 空状态(非手动 非自动 非急停 非设置)
	bIdle:					BOOL;// 设备空闲
	bBreakpoint:			BOOL;// 断点模式
	eLanguage:				E_Language;// 当前语言
END_STRUCT
END_TYPE

// System/DUTs/ST_SystemOutput
TYPE ST_SystemOutput :
STRUCT
	bBuzzer:				BOOL;// 蜂鸣器
	bLightRed:				BOOL;// 红色报警指示灯
	bLightGreen:			BOOL;// 绿色运行指示灯
	bLightYellow:			BOOL;// 黄色停止指示灯
END_STRUCT
END_TYPE

// System/DUTs/ST_SystemStation
TYPE ST_SystemStation :
STRUCT
	arrName:				ARRAY[0..E_Language.MaxCount] OF WSTRING;// 工站名称
	arrInfo:				ARRAY[0..E_Language.MaxCount] OF WSTRING;// 信息
	arrStepHistory:			ARRAY[0..9] OF ST_SystemStationHistory;// 历史步
	iStepPrev:				UINT;// 上一步
	iStepNow:				UINT;// 当前步
	iStepNext:				UINT;// 下一步(当设备正常运行时,将下步赋值给当前步)
END_STRUCT
END_TYPE

// System/DUTs/ST_SystemStationHistory
TYPE ST_SystemStationHistory :
STRUCT
	arrName:					ARRAY[0..E_Language.MaxCount] OF	WSTRING;
	iStep:						UINT;
	arrInfo:					ARRAY[0..E_Language.MaxCount] OF	WSTRING;
END_STRUCT
END_TYPE

// System/DUTs/ST_TriggerMode
TYPE ST_TriggerMode :
STRUCT
	bAuto:				BOOL;// 自动
	bManual:			BOOL;// 手动
END_STRUCT
END_TYPE

// TcpIp/DUTs/E_TcpIpClientCmd
{attribute 'qualified_only'}
{attribute 'strict'}
TYPE E_TcpIpClientCmd :
(
	None:=0,
	Connect,
	Disconnect,
	Read,
	Write,
	Reset
);
END_TYPE

// TcpIp/DUTs/ST_TcpIpClient
TYPE ST_TcpIpClient :
STRUCT
	ID:								BYTE;
	sName:							WSTRING;// 实例名称(只读)
	stContorl:						ST_TcpIpClientControl;// 控制
	stStatus:						ST_TcpIpClientStatus;// 状态
	sSendData:						STRING(1000);// 发送数据
	sReceiveData:					STRING(1000);// 接收数据
	arrInfo:						ARRAY[0..E_Language.MaxCount] OF ST_TcpIpClientInfo;// 多语言信息
END_STRUCT
END_TYPE

// TcpIp/DUTs/ST_TcpIpClientControl
TYPE ST_TcpIpClientControl :
STRUCT
	stConnect:						ST_TriggerMode;// 连接
	stSend:							ST_TriggerMode;// 发送
	stReceive:						ST_TriggerMode;// 接收
	stClose:						ST_TriggerMode;// 关闭
END_STRUCT
END_TYPE

// TcpIp/DUTs/ST_TcpIpClientInfo
TYPE ST_TcpIpClientInfo :
STRUCT
	sName:					WSTRING;// 名称
	sConnectError:			WSTRING;// 连接错误
	sSendError:				WSTRING;// 发送错误
	sReceiveError:			WSTRING;// 接收错误
	sCloseError:			WSTRING;// 关闭错误			
END_STRUCT
END_TYPE

// TcpIp/DUTs/ST_TcpIpClientStatus
TYPE ST_TcpIpClientStatus :
STRUCT
	bConnected:				BOOL;// 已连接
	bSent:					BOOL;// 发送完成
	bReceived:				BOOL;// 接收完成
	bClosed:				BOOL;// 已关闭
	bSending:				BOOL;// 发送中
	bReceiving:				BOOL;// 接收中
	bConnecting:			BOOL;// 连接中
	bClosing:				BOOL;// 关闭中
	bError:					BOOL;// 错误状态 
	bErrorConnect:			BOOL;// 连接错误
	bErrorSend:				BOOL;// 发送错误
	bErrorReceive:			BOOL;// 接收错误
	bErrorClose:			BOOL;// 关闭错误
END_STRUCT
END_TYPE

// TcpIp/DUTs/ST_TcpIpData
TYPE ST_TcpIpData :
STRUCT
	sServerIp:						STRING;// 服务器地址
	iServerPort:					UINT;// 服务器端口号
END_STRUCT
END_TYPE

// Yield/DUTs/ST_Yield
TYPE ST_Yield :
STRUCT
	stControl:				ST_YieldControl;
END_STRUCT
END_TYPE

// Yield/DUTs/ST_YieldControl
TYPE ST_YieldControl :
STRUCT
	bOk:				BOOL;
	bNG:				BOOL;
	bTOSS:				BOOL;
	bClear:				BOOL;
	bAutoClear:			BOOL;
END_STRUCT
END_TYPE

// Yield/DUTs/ST_YieldData
TYPE ST_YieldData :
STRUCT
	iAll:				INT;// 总产能
	iNG:				INT;// 不良产能
	iOK:				INT;// 合格产能
	iTOSS:				INT;// 抛料产能
	fNgPercentage:		REAL;// 不良率
	fOkPercentage:		REAL;// 合格率
	fTOSSPercentage:	REAL;// 抛料率
END_STRUCT
END_TYPE

// Version/Global_Version
{attribute 'TcGenerated'}
{attribute 'no-analysis'}
{attribute 'linkalways'}
// This function has been automatically generated from the project information.
VAR_GLOBAL CONSTANT
	{attribute 'const_non_replaced'}
	stLibVersion_MachineManage : ST_LibVersion := (iMajor := 1, iMinor := 3, iBuild := 0, iRevision := 0, nFlags := 0, sVersion := '1.3.0.0');
END_VAR

// GVL
{attribute 'qualified_only'}
{attribute'hide'}
VAR_GLOBAL
	bWindowsCmdLock:					BOOL;
	bFileErrorLogLock:					BOOL;
	sErrorInfo:							STRING(2000);
	sErrorInfoTemp:						WSTRING(2000);								
	FbErrorLog:							FB_FileHelper;
END_VAR

// GVL_Data_P
VAR_GLOBAL PERSISTENT
	G_arrAxisData:			ARRAY[0..20] OF ST_AxisData;
	G_arrCylinderData:		ARRAY[0..50] OF ST_CylinderData;
END_VAR

// GVL_P
VAR_GLOBAL
	G_stSystem:				ST_System;
	G_stError:				ST_Error;
	
	G_arrStation:			ARRAY[0..20] OF ST_SystemStation;
	
	G_arrCylinder:			ARRAY[0..50] OF ST_Cylinder;
	G_arrAxis:				ARRAY[0..20] OF ST_Axis;
	
	G_arrFbAxis:			ARRAY[0..20] OF FB_Axis;
	G_arrFbCylinder:		ARRAY[0..50] OF FB_Cylinder;
END_VAR

// Axis/POUs/FB_Axis
FUNCTION_BLOCK FB_Axis
VAR_INPUT
	Axis:					 	REFERENCE TO  ST_Axis;// 轴控制集合
	Data:						REFERENCE TO  ST_AxisData;// 轴数据
	Error:						REFERENCE TO  ST_Error;// 报警集合
	System:						REFERENCE TO  ST_System;// 系统集合
END_VAR
VAR_OUTPUT
END_VAR
VAR
	_mcRest:					MC_Reset;// 轴复位
	_mcStop:					MC_Stop;// 轴停止
	_mcPower:					MC_Power;// 轴使能
	_mcJog:						MC_Jog;// 轴点动
	_mcHome:					MC_Home;// 轴回零
	_mcMoveAbsolute:			MC_MoveAbsolute;// 轴定位
	_mcMoveRelative:			MC_MoveRelative;// 轴相对定位
	_bHomeSatrt:				BOOL;// 启动回零信号
	_bStartAbs:					BOOL;// 启动绝对定位信号
	_bStartRel:					BOOL;// 启动相对定位信号
	_tonHome:					TON;// 回零时间
	_i:							INT;
	_rHomeBusy:					R_TRIG;// 回零中
	_rAbsBusy:					R_TRIG;// 绝对定位中
	_rRelBusy:					R_TRIG;// 相对定位中
	_rHomeDone:					R_TRIG;// 回零完成
	_fPowered:					F_TRIG;// 使能
	_rAbs:						F_TRIG;
	_rRel:						F_TRIG;
	_arrFbError:				ARRAY[0..10]OF FB_ErrorTag;// 报警模块
	
	_iHomeDirection:			INT;// 1: 为正向回零 -1:为反向回零

	_fbMemoryLag:				FB_MemoryLag;// 记忆
	
	_rStop:					 	R_TRIG;
	_bFirstDryRun:				BOOL:=TRUE;
	
	_tonHomeV:					TON;// 速度回零模式计时
	
	_fMoveRelTemp:				LREAL;
	_teach:						TON;// 手动示教延迟
	_bMoveMemory:				BOOL;
	
END_VAR

// 当前名称
Axis.sName:=Axis.arrInfo[System.stMode.eLanguage].sName;

IF Axis.stLock.bShield THEN
	RETURN;
END_IF


// 轴运行中
Axis.Axis_REF.ReadStatus();
Axis.stStatus.bMoving:=Axis.Axis_REF.Status.Moving OR _mcJog.Busy OR _mcHome.Busy OR _mcMoveAbsolute.Busy OR _mcMoveRelative.Busy;


IF _bFirstDryRun THEN
	A_Init();
END_IF

A_ControlRest();

A_Power();

A_Rest();

A_Home();

A_Stop();

A_Jog();

A_MoveAbsolute();

A_MoveRelative();

A_Error();

A_Memory();

A_Teach();

_bFirstDryRun:=FALSE;

ACTION A_ControlRest:
{attribute'hide'}

// 轴控制状态复位
IF System.stMode.stDeviceRest.bAuto THEN
	Axis.stControl.stHome.bAuto:=FALSE;
	Axis.stControl.stMovePosition.stStartAbs.bAuto:=FALSE;
	Axis.stControl.stMovePosition.stStartRel.bAuto:=FALSE;
	Axis.stControl.stJog.stNegative.bAuto:=FALSE;
	Axis.stControl.stJog.stPositive.bAuto:=FALSE;
	Axis.stControl.stReset.bAuto:=FALSE;
	Axis.stControl.stStop.bAuto:=FALSE;
	Axis.stControl.stClosePower.bAuto:=FALSE;
	Axis.stControl.stTeach.bAuto:=FALSE;
	Axis.stControl.stMoveMemory.bAuto:=FALSE;
END_IF;
IF System.stMode.stDeviceRest.bManual THEN
	Axis.stControl.stHome.bManual:=FALSE;
	Axis.stControl.stMovePosition.stStartAbs.bManual:=FALSE;
	Axis.stControl.stMovePosition.stStartRel.bManual:=FALSE;
	Axis.stControl.stJog.stNegative.bManual:=FALSE;
	Axis.stControl.stJog.stPositive.bManual:=FALSE;
	Axis.stControl.stReset.bManual:=FALSE;
	Axis.stControl.stStop.bManual:=FALSE;
	Axis.stControl.stClosePower.bManual:=FALSE;
	Axis.stControl.stTeach.bManual:=FALSE;
	Axis.stControl.stMoveMemory.bManual:=FALSE;
END_IF;
END_ACTION

ACTION A_Error:
{attribute'hide'}

// 轴错误
Axis.stStatus.bError:=Axis.Axis_REF.Status.Error;
// 轴错误代码
Axis.stStatus.iErrorID:=Axis.Axis_REF.NcToPlc.ErrorCode;
// 功能块报警
_arrFbError[0](
	Error:=Error , 
	System:=System , 
	Enable:=Axis.Axis_REF.NcToPlc.ErrorCode<>0 , 
	Message:= , 
	Level:= 2,
	Position:=WCONCAT("FB_Axis:",Axis.arrInfo[System.stMode.eLanguage].sName),
	Erroring=>Axis.stStatus.bErrorFB,
	ID:=Axis.ID,
	Category:=E_ErrorCategory.Axis,
	InfoIndex:=0);
IF _arrFbError[0].Erroring OR _bFirstDryRun THEN
	FOR _i:=0 TO E_Language.MaxCount BY 1 DO
		_arrFbError[0].Language[_i]:=WCONCAT(Axis.arrInfo[_i].sName,WCONCAT(Axis.arrInfo[_i].sFbErrorInfo,UDINT_TO_WSTRING(Axis.stStatus.iErrorID)));
	END_FOR
END_IF

// 负极限报警
_arrFbError[1](
	Error:=Error , 
	System:=System , 
	Enable:=Axis.stInput.bNegative AND NOT (Data.stMode.iHomeMode=0 AND _iHomeDirection=-1 AND _mcHome.Busy) , 
	Message:= , 
	Level:= 2,
	Position:=WCONCAT("FB_Axis:",Axis.arrInfo[System.stMode.eLanguage].sName),
	Erroring=>Axis.stStatus.bErrorNegative,
	ID:=Axis.ID,
	Category:=E_ErrorCategory.Axis,
	InfoIndex:=1);

// 正极限报警
_arrFbError[2](
	Error:=Error , 
	System:=System , 
	Enable:=Axis.stInput.bPositive AND NOT (Data.stMode.iHomeMode=0 AND _iHomeDirection=1 AND _mcHome.Busy) , 
	Message:=, 
	Level:= 2,
	Position:=WCONCAT("FB_Axis:",Axis.arrInfo[System.stMode.eLanguage].sName),
	Erroring=>Axis.stStatus.bErrorPositive,
	ID:=Axis.ID,
	Category:=E_ErrorCategory.Axis,
	InfoIndex:=2);

// 回零超时
_arrFbError[3](
	Error:=Error , 
	System:=System , 
	Enable:=_mcHome.Busy , 
	Message:= , 
	Level:= 4,
	Position:=WCONCAT("FB_Axis:",Axis.arrInfo[System.stMode.eLanguage].sName),
	Erroring=>Axis.stStatus.bErrorHome,
	ErrorTime:=T#60S,
	ID:=Axis.ID,
	Category:=E_ErrorCategory.Axis,
	InfoIndex:=3);
END_ACTION

ACTION A_Home:
{attribute'hide'}

// 轴回零
_bHomeSatrt:=(Axis.stControl.stHome.bManual AND System.stMode.stDeviceEnable.bManual) OR (Axis.stControl.stHome.bAuto AND System.stMode.stDeviceEnable.bAuto);
_mcHome.Execute:=_bHomeSatrt AND NOT Axis.stLock.bHome AND NOT Axis.stLock.bAll;

// 计算回零方向
IF _mcHome.Busy AND _iHomeDirection=0 AND ABS(Axis.Axis_REF.NcToPlc.ActVelo)>0.5 THEN
	_iHomeDirection:=SEL(Axis.Axis_REF.NcToPlc.ActPos<0,-1,1);
END_IF
IF (Axis.stControl.stReset.bManual AND System.stMode.stDeviceEnable.bManual) OR (Axis.stControl.stReset.bAuto AND System.stMode.stDeviceEnable.bAuto) OR System.stInput.bReset OR _mcHome.Done THEN
	_iHomeDirection:=0;
	_mcHome.bCalibrationCam:=FALSE;
END_IF

// 回零方式判断
CASE Data.stMode.iHomeMode OF
	0:// 按原点信号回零
		_mcHome.HomingMode:=MC_DefaultHoming;
		CASE _iHomeDirection OF
			-1:// 反向回零
				_mcHome.bCalibrationCam:=Axis.stInput.bNegative;
			1:// 正向回零
				_mcHome.bCalibrationCam:=Axis.stInput.bPositive;
		END_CASE
	1:// 力矩反馈回零
		_mcHome.HomingMode:=MC_DefaultHoming;
		IF ABS(Axis.Axis_REF.NcToPlc.ActVelo) <Data.iSetHomeVelocity AND ABS(Data.stTorque.iGetTorque) > Data.stTorque.iSetTorque * 0.8 AND NOT _mcHome.bCalibrationCam AND _iHomeDirection<>0  THEN
			_mcHome.bCalibrationCam:= TRUE;
		END_IF
		IF _mcHome.bCalibrationCam THEN
			IF  _iHomeDirection<0 AND  Axis.Axis_REF.NcToPlc.ActPos>=-9999999995 AND Axis.Axis_REF.NcToPlc.ActPos<0 THEN
				_mcHome.bCalibrationCam:=FALSE;
			END_IF
			IF _iHomeDirection>0 AND Axis.Axis_REF.NcToPlc.ActPos<=9999999995 AND  Axis.Axis_REF.NcToPlc.ActPos>0 THEN
				_mcHome.bCalibrationCam:=FALSE;
			END_IF
		END_IF
	2:// 设置当前位置为原点
		_mcHome.HomingMode:=MC_Direct;
	3:// 速度回零模式
		_mcHome.HomingMode:=MC_DefaultHoming;
		_tonHomeV(IN:=ABS(Axis.Axis_REF.NcToPlc.ActVelo) <Data.iSetHomeVelocity AND _mcHome.Busy AND NOT _mcHome.bCalibrationCam AND _iHomeDirection<>0 , PT:=T#1S , Q=> , ET=> );
		IF _tonHomeV.Q THEN
			_mcHome.bCalibrationCam:= TRUE;
		END_IF;
		IF _mcHome.bCalibrationCam THEN
			IF  _iHomeDirection<0 AND  Axis.Axis_REF.NcToPlc.ActPos>=-9999999995 AND Axis.Axis_REF.NcToPlc.ActPos<0 THEN
				_mcHome.bCalibrationCam:=FALSE;
			END_IF;
			IF _iHomeDirection>0 AND Axis.Axis_REF.NcToPlc.ActPos<=9999999995 AND  Axis.Axis_REF.NcToPlc.ActPos>0 THEN
				_mcHome.bCalibrationCam:=FALSE;
			END_IF;
		END_IF;
END_CASE

_mcHome(
	Axis:= Axis.Axis_REF, 
	Execute:= , 
	Position:= DEFAULT_HOME_POSITION, // 使用虚拟轴中参数
	HomingMode:= ,
	BufferMode:= , 
	Options:= , 
	bCalibrationCam:= , 
	Done=> , 
	Busy=> , 
	Active=> , 
	CommandAborted=> , 
	Error=> , 
	ErrorID=> );
	
//轴回零中
Axis.stStatus.bHoming:=_mcHome.Busy;
//回零完成
_rHomeBusy(CLK:=_mcHome.Busy , Q=> );
IF _rHomeBusy.Q OR 
	System.stInput.bReset OR// 总复位
	(Axis.stControl.stReset.bManual AND System.stMode.stDeviceEnable.bManual) OR // 手动复位
	(Axis.stControl.stReset.bAuto AND System.stMode.stDeviceEnable.bAuto) OR // 自动复位
	(System.stMode.bAuto AND (System.stMode.arrAlarm[1] OR System.stMode.arrAlarm[2])) THEN// 自动状态 1,2级报警
		
	Axis.stStatus.bHomeDone:=FALSE;
END_IF;
_rHomeDone(CLK:=_mcHome.Done , Q=> );
IF _rHomeDone.Q THEN
	Axis.stStatus.bHomeDone:=TRUE;
END_IF;
END_ACTION

ACTION A_Init:
{attribute'hide'}

Axis.arrInfo[E_Language.Chinese].sFbErrorInfo:=":功能模块错误代码:";
Axis.arrInfo[E_Language.Chinese].sHomeInfo:=":回零超时!(此消息只做提醒)";
Axis.arrInfo[E_Language.Chinese].sNegativeInfo:=":碰负极限 请手动移离极限后 重新初始化!";
Axis.arrInfo[E_Language.Chinese].sPositiveInfo:=":碰正极限 请手动移离极限后 重新初始化!";
Axis.arrInfo[E_Language.Chinese].sMemoryPos:=":记忆位置和当前位置不符合";

Axis.arrInfo[E_Language.English].sFbErrorInfo:=": function module error code :";
Axis.arrInfo[E_Language.English].sHomeInfo:=": back to zero timeout!";
Axis.arrInfo[E_Language.English].sNegativeInfo:=": hits the negative limit";
Axis.arrInfo[E_Language.English].sPositiveInfo:=": hits the positive limit";
Axis.arrInfo[E_Language.English].sMemoryPos:=": The memory location does not match the current location";

Axis.arrInfo[E_Language.Vietnamese].sFbErrorInfo:=": mã lỗi môđun chức năng :";
Axis.arrInfo[E_Language.Vietnamese].sHomeInfo:=": Quay lại thời gian không!";
Axis.arrInfo[E_Language.Vietnamese].sNegativeInfo:=": Chạm đến giới hạn tiêu cực";
Axis.arrInfo[E_Language.Vietnamese].sPositiveInfo:=": Chạm vào giới hạn tích cực";
Axis.arrInfo[E_Language.Vietnamese].sMemoryPos:=": vị trí ghi nhớ và vị trí hiện tại không phù hợp";

Axis.arrInfo[E_Language.Hindi].sFbErrorInfo:=": फ़ंक्शन मॉड्यूल त्रुटि कोड::";
Axis.arrInfo[E_Language.Hindi].sHomeInfo:=": शून्य मध्यांतर में वापस";
Axis.arrInfo[E_Language.Hindi].sNegativeInfo:=": सीमा मारो";
Axis.arrInfo[E_Language.Hindi].sPositiveInfo:=": सही सीमा मारो";
Axis.arrInfo[E_Language.Hindi].sMemoryPos:=": स्मृति की स्थिति वर्तमान स्थिति से मेल नहीं खाती है ";

FOR _i:=0 TO E_Language.MaxCount BY 1 DO
	_arrFbError[1].Language[_i]:=WCONCAT(Axis.arrInfo[_i].sName, Axis.arrInfo[_i].sNegativeInfo);
	_arrFbError[2].Language[_i]:=WCONCAT(Axis.arrInfo[_i].sName ,Axis.arrInfo[_i].sPositiveInfo);
	_arrFbError[3].Language[_i]:=WCONCAT(Axis.arrInfo[_i].sName, Axis.arrInfo[_i].sHomeInfo);
	
	_fbMemoryLag.Language[_i]:=WCONCAT(Axis.arrInfo[_i].sName ,Axis.arrInfo[_i].sMemoryPos);
END_FOR
END_ACTION

ACTION A_Jog:
{attribute'hide'}

// 轴点动
_mcJog.JogForward:=((System.stMode.stDeviceEnable.bAuto AND Axis.stControl.stJog.stPositive.bAuto)  OR (System.stMode.stDeviceEnable.bManual AND Axis.stControl.stJog.stPositive.bManual)) AND NOT Axis.stLock.bJogPositive AND NOT Axis.stLock.bAll;
_mcJog.JogBackwards:=((System.stMode.stDeviceEnable.bAuto AND Axis.stControl.stJog.stNegative.bAuto)  OR (System.stMode.stDeviceEnable.bManual AND Axis.stControl.stJog.stNegative.bManual)) AND NOT  Axis.stLock.bJogNegative AND NOT Axis.stLock.bAll;

_mcJog(
	Axis:= Axis.Axis_REF, 
	JogForward:= , 
	JogBackwards:= , 
	Mode:= MC_JOGMode_CONTINOUS, 
	Position:= , 
	Velocity:= Data.fJogVelocity, 
	Acceleration:= Data.fJogAccelerated, 
	Deceleration:= Data.fJogDeceleration, 
	Jerk:= , 
	Done=> , 
	Busy=> , 
	Active=> , 
	CommandAborted=> , 
	Error=> , 
	ErrorID=> );
END_ACTION

ACTION A_Memory:
{attribute'hide'}

_fbMemoryLag(
	Value:=Axis.Axis_REF.NcToPlc.ActPos, 
	Lag:=0.5 , 
	System:=System , 
	Error:=Error , 
	Message:= , 
	Position:=WCONCAT("FB_Axis:",Axis.arrInfo[System.stMode.eLanguage].sName) , 
	Erroring=>Axis.stStatus.bMemoryPos,
	ID:=Axis.ID,
	Category:=E_ErrorCategory.Axis,
	InfoIndex:=20,
	MemoryValue=>Data.fMemoryPosition );
END_ACTION

ACTION A_MoveAbsolute:
{attribute'hide'}

// 轴绝对定位
_bMoveMemory:=((System.stMode.stDeviceEnable.bAuto AND Axis.stControl.stMoveMemory.bAuto) OR (System.stMode.stDeviceEnable.bManual AND Axis.stControl.stMoveMemory.bManual)) AND Axis.stStatus.bMemoryPos;
_bStartAbs:=(System.stMode.stDeviceEnable.bAuto AND Axis.stControl.stMovePosition.stStartAbs.bAuto) OR (System.stMode.stDeviceEnable.bManual AND Axis.stControl.stMovePosition.stStartAbs.bManual);


_mcMoveAbsolute.Execute:=( _bStartAbs OR _bMoveMemory) AND NOT Axis.stLock.arrMovePosition[Axis.stControl.stMovePosition.iIndex] AND NOT Axis.stLock.bAll AND NOT Axis.stLock.bMoveAbsAll;

_mcMoveAbsolute(
	Axis:= Axis.Axis_REF, 
	Execute:= , 
	Position:=SEL(_bMoveMemory,Data.arrMovePosition[Axis.stControl.stMovePosition.iIndex],Data.fMemoryPosition), 
	Velocity:= Data.arrMoveVelocity[Axis.stControl.stMovePosition.iIndex], 
	Acceleration:=Data.arrMoveAccelerated[Axis.stControl.stMovePosition.iIndex], 
	Deceleration:= Data.arrMoveDeceleration[Axis.stControl.stMovePosition.iIndex], 
	Jerk:= , 
	BufferMode:= , 
	Options:= , 
	Done=> , 
	Busy=> , 
	Active=> , 
	CommandAborted=> , 
	Error=> , 
	ErrorID=> );
	
Axis.stStatus.bMoveAbsDone:=M_GetAbsDone(Axis.stControl.stMovePosition.iIndex);
END_ACTION

ACTION A_MoveRelative:
{attribute'hide'}

// 轴相对定位
_bStartRel:=(System.stMode.stDeviceEnable.bAuto AND Axis.stControl.stMovePosition.stStartRel.bAuto) OR (System.stMode.stDeviceEnable.bManual AND Axis.stControl.stMovePosition.stStartRel.bManual);
_mcMoveRelative.Execute:= _bStartRel AND NOT Axis.stLock.arrMovePosition[Axis.stControl.stMovePosition.iIndex]  AND NOT Axis.stLock.bAll AND NOT Axis.stLock.bMoveRelAll;

_rRelBusy(CLK:=_mcMoveRelative.Execute , Q=> );
IF  _rRelBusy.Q AND NOT Axis.stStatus.bMoving THEN
	_fMoveRelTemp:=Axis.Axis_REF.NcToPlc.ActPos;
END_IF

_mcMoveRelative(
	Axis:=Axis.Axis_REF , 
	Execute:= , 
	Distance:=Data.arrMovePosition[Axis.stControl.stMovePosition.iIndex] , 
	Velocity:=Data.arrMoveVelocity[Axis.stControl.stMovePosition.iIndex] , 
	Acceleration:=Data.arrMoveAccelerated[Axis.stControl.stMovePosition.iIndex] , 
	Deceleration:=Data.arrMoveDeceleration[Axis.stControl.stMovePosition.iIndex] , 
	Jerk:= , 
	BufferMode:= , 
	Options:= , 
	Done=> , 
	Busy=> , 
	Active=> , 
	CommandAborted=> , 
	Error=> , 
	ErrorID=> );
	
Axis.stStatus.bMoveRelDone:=M_GetRelDone(Axis.stControl.stMovePosition.iIndex);
END_ACTION

ACTION A_Power:
{attribute'hide'}

// 轴上电控制
_mcPower.Enable:=(System.stMode.bAuto OR System.stMode.bManual) AND NOT System.stMode.bEStop;
IF System.stMode.stDeviceEnable.bManual AND Axis.stControl.stClosePower.bManual THEN
	_mcPower.Enable:=FALSE;
END_IF;

_mcPower(
	Axis:=Axis.Axis_REF , 
	Enable:= , 
	Enable_Positive:= TRUE, 
	Enable_Negative:= TRUE, 
	Override:= 100.0, 
	BufferMode:= , 
	Options:= , 
	Status=> , 
	Busy=> , 
	Active=> , 
	Error=> , 
	ErrorID=> ); 
	
	
_fPowered(CLK:=_mcPower.Busy , Q=> );
IF NOT _mcPower.Error AND _fPowered.Q THEN
	Axis.stStatus.bPowered:=TRUE;
END_IF;
IF NOT _mcPower.Enable OR _mcPower.Error THEN
	Axis.stStatus.bPowered:=FALSE;
END_IF;
END_ACTION

ACTION A_Rest:
{attribute'hide'}

// 轴复位
_mcRest(
	Axis:= Axis.Axis_REF, 
	Execute:=(Axis.stControl.stReset.bManual AND System.stMode.stDeviceEnable.bManual) OR (Axis.stControl.stReset.bAuto AND System.stMode.stDeviceEnable.bAuto) OR System.stInput.bReset , 
	Done=> , 
	Busy=> , 
	Error=> , 
	ErrorID=> );
END_ACTION

ACTION A_Stop:
{attribute'hide'}

_rStop(CLK:=System.stMode.bStop , Q=> );

// 轴停止控制
IF  Axis.stStatus.bError OR// 轴错误
	_rStop.Q OR// 停止状态 轴立即停止
	System.stMode.bEStop OR// 急停状态
	(Axis.stControl.stStop.bAuto AND System.stMode.stDeviceEnable.bAuto) OR // 自动停止
	(Axis.stControl.stStop.bManual AND System.stMode.stDeviceEnable.bManual) OR // 手动停止
	(Axis.stInput.bNegative AND NOT Axis.stControl.stJog.stPositive.bManual AND NOT (Data.stMode.iHomeMode=0 AND _iHomeDirection=-1 AND _mcHome.Busy)) OR// 碰负极限
	(Axis.stInput.bPositive AND NOT Axis.stControl.stJog.stNegative.bManual AND NOT (Data.stMode.iHomeMode=0 AND _iHomeDirection=1 AND _mcHome.Busy)) THEN // 碰正极限
	_mcStop.Execute:=TRUE;
ELSE
	_mcStop.Execute:=FALSE;
END_IF;
_mcStop(
	Axis:= Axis.Axis_REF, 
	Execute:=, 
	Deceleration:=900000000, 
	Jerk:= , 
	Options:= , 
	Done=> , 
	Busy=> , 
	Active=> , 
	CommandAborted=> , 
	Error=> , 
	ErrorID=> );
END_ACTION

ACTION A_Teach:
{attribute'hide'}
_teach(IN:=(System.stMode.stDeviceEnable.bManual AND Axis.stControl.stTeach.bManual) , PT:=T#1S , Q=> , ET=> );

IF (System.stMode.stDeviceEnable.bAuto AND Axis.stControl.stTeach.bAuto) OR _teach.Q THEN
	Data.arrMovePosition[Axis.stControl.stMovePosition.iIndex]:=Axis.Axis_REF.NcToPlc.ActPos;
END_IF;
END_ACTION

METHOD M_GetAbsDone : BOOL
VAR_INPUT
	Index:					UINT;
END_VAR
M_GetAbsDone:=(ABS(Axis.Axis_REF.NcToPlc.ActPos-Data.arrMovePosition[Index])<=ABS(Data.iSetMoveFluctuation)) AND NOT Axis.stStatus.bMoving;
END_METHOD

METHOD M_GetRelDone : BOOL
VAR_INPUT
	Index:					UINT;
END_VAR
VAR
	temp:					LREAL;
END_VAR
temp:=_fMoveRelTemp+Data.arrMovePosition[Index];
M_GetRelDone:=(ABS(Axis.Axis_REF.NcToPlc.ActPos-temp)<=ABS(Data.iSetMoveFluctuation)) AND NOT Axis.stStatus.bMoving;
END_METHOD

METHOD M_Home : BOOL
VAR_INPUT
END_VAR
IF NOT  Axis.stStatus.bMoving AND NOT Axis.stStatus.bHomeDone THEN
	Axis.stControl.stHome.bAuto:=TRUE;
END_IF;

IF Axis.stStatus.bMoving OR Axis.stStatus.bHomeDone  THEN
	Axis.stControl.stHome.bAuto:=FALSE;
END_IF;

M_Home:=Axis.stStatus.bHomeDone;
END_METHOD

METHOD M_Jog 
VAR_INPUT
	Command:					INT;// -1:反转; 0:停止; 1:正转; 
END_VAR
CASE Command OF
	-1:
		Axis.stControl.stJog.stPositive.bAuto:=FALSE;
		Axis.stControl.stJog.stNegative.bAuto:=TRUE;
	0:
		Axis.stControl.stJog.stPositive.bAuto:=FALSE;
		Axis.stControl.stJog.stNegative.bAuto:=FALSE;
	1:
		Axis.stControl.stJog.stPositive.bAuto:=TRUE;
		Axis.stControl.stJog.stNegative.bAuto:=FALSE;
END_CASE;
END_METHOD

METHOD M_MoveAbs : BOOL
VAR_INPUT
	Index:					UINT;// 定位索引
END_VAR
IF System.stMode.bStop THEN
	M_MoveAbs:=FALSE;
	RETURN;
END_IF

Axis.stControl.stMovePosition.iIndex:=Index;
IF NOT Axis.stStatus.bMoving  THEN
	Axis.stControl.stMovePosition.stStartAbs.bAuto:=TRUE;
END_IF;
IF Axis.stStatus.bMoving OR M_GetAbsDone(Index)THEN
	Axis.stControl.stMovePosition.stStartAbs.bAuto:=FALSE;
END_IF;

M_MoveAbs:=M_GetAbsDone(Index);
END_METHOD

METHOD M_MoveRel : BOOL
VAR_INPUT
	Index:					UINT;// 定位索引
END_VAR
IF  System.stMode.bStop THEN
	M_MoveRel:=FALSE;
	RETURN;
END_IF

Axis.stControl.stMovePosition.iIndex:=Index;
IF NOT Axis.stStatus.bMoving THEN
	Axis.stControl.stMovePosition.stStartRel.bAuto:=TRUE;
END_IF;
IF Axis.stStatus.bMoving OR M_GetRelDone(Index) THEN
	Axis.stControl.stMovePosition.stStartRel.bAuto:=FALSE;
END_IF;

M_MoveRel:=M_GetRelDone(Index);
END_METHOD

END_FUNCTION_BLOCK

// Error/POUs/FB_ErrorTag
FUNCTION_BLOCK FB_ErrorTag
VAR_INPUT
	System:					REFERENCE TO ST_System;
	Error:					REFERENCE TO ST_Error;
	ID:						BYTE;// ID 从50开始(生成ErrorCode使用 如无相关需求可忽略)
	Category:				E_ErrorCategory;// 报警类别(生成ErrorCode使用 如无相关需求可忽略)
	InfoIndex:				BYTE;// 从50开始(生成ErrorCode使用 如无相关需求可忽略)
	Enable:					BOOL;// 报警触发
	Message:				WSTRING;// 报警内容(中文)
	Level:					BYTE:=1;// 报警等级
	Position:				WSTRING;// 错误发生位置
	ErrorTime:				TIME:=T#0S;// 报警延迟
	Language:				ARRAY[0..E_Language.MaxCount] OF WSTRING;//	其他语言集合
END_VAR
VAR_OUTPUT
	Erroring:				BOOL;
	ErrorCode:				DWORD;
END_VAR
VAR
	_i:						INT;
	_iCyclic:				INT;
	_iRunNow:				INT;
	_tonError:				TON;
	_iTemp:					INT;
	_stNullInfo:			ST_ErrorInfo;
	_rTRIG:					R_TRIG;
	
	_iRun:					UINT;
	
	_iErrorCode:			DWORD;
	_pErrorCode:			POINTER TO BYTE;
	_arrErrorList:			ARRAY[0..10] OF WSTRING;
END_VAR

IF  _iCyclic<10 THEN
	_iCyclic:=_iCyclic+1;
	RETURN;
END_IF;

_pErrorCode:= ADR(_iErrorCode);
_pErrorCode[3]:=TO_BYTE(Category);
_pErrorCode[2]:=ID;
_pErrorCode[1]:=TO_BYTE(Level);
_pErrorCode[0]:=InfoIndex;

_tonError(IN:=Enable , PT:=ErrorTIME , Q=> , ET=> );

IF System.stInput.bReset OR System.stInput.bResetAlarm THEN
	ErrorCode:=0;
	Erroring:=FALSE;
	_iRunNow:=0;
END_IF;

// 记录当前报警
CASE _iRunNow OF
	0:
		_rTRIG.CLK:=FALSE;
		IF _tonError.Q AND NOT Erroring THEN
			_iRunNow:=100;
		END_IF;
	100:
		System.stMode.arrAlarm[Level]:=TRUE;
		Erroring:=TRUE;
		ErrorCode:=_iErrorCode;
		_iRunNow:=200;
	200:
		_rTRIG.CLK:=TRUE;
		FOR _i:=0 TO Error.stNow.iCount BY 1 DO
			IF NOT Error.stNow.arrInfo[_i].bStatus THEN
				Error.stNow.arrInfo[_i].sSystemDate:=System.stSystemDate.sNow;
				Error.stNow.arrInfo[_i].bStatus:=TRUE;
				Error.stNow.arrInfo[_i].sLevel:=TO_STRING(Level);
				Error.stNow.arrInfo[_i].sPosition:=Position;
				Error.stNow.arrInfo[_i].arrMessage:=Language;
				Error.stNow.arrInfo[_i].iErrorCode:=ErrorCode;
				IF Message<>"" THEN
					Error.stNow.arrInfo[_i].arrMessage[E_Language.Chinese]:=Message;
				END_IF;
				_iTemp:=_i;
				EXIT;
			END_IF;
		END_FOR;
		_iRunNow:=300;
	300:
		IF Level=5 AND NOT System.stInput.bReset AND NOT System.stInput.bResetAlarm  THEN
			System.stMode.arrAlarm[5]:=TRUE;
		END_IF;
		IF NOT Enable THEN
			_iRunNow:=400;
		END_IF;
	400:
		IF Level=5 THEN
			Erroring:=FALSE;
			Error.stNow.arrInfo[_iTemp]:=_stNullInfo;
			System.stMode.arrAlarm[5]:=FALSE;
		END_IF;
		_iRunNow:=0;
END_CASE;

// 记录历史报警
_rTRIG(CLK:= , Q=> );
IF _rTRIG.Q THEN
	FOR _i:=Error.stHistory.iCount TO 1 BY -1 DO
		Error.stHistory.arrInfo[_i]:=Error.stHistory.arrInfo[_i-1];
	END_FOR;
	Error.stHistory.arrInfo[0].bStatus:=TRUE;
	Error.stHistory.arrInfo[0].sSystemDate:=System.stSystemDate.sNow;
	Error.stHistory.arrInfo[0].arrMessage:=Language;
	Error.stHistory.arrInfo[0].sLevel:=TO_STRING(Level);
	Error.stHistory.arrInfo[0].sPosition:=Position;
	Error.stHistory.arrInfo[0].iErrorCode:=ErrorCode;
	IF Message<>"" THEN
		Error.stHistory.arrInfo[0].arrMessage[E_Language.Chinese]:=Message;
	END_IF;
END_IF;


CASE _iRun OF
	0:
		IF Error.bSaveErrorList THEN
			_iRun:=100;
		END_IF
	100:
		IF NOT GVL.bFileErrorLogLock THEN
			GVL.bFileErrorLogLock:=TRUE;
			_iRun:=200;
		END_IF
	200:
		IF  Level>3 THEN
			 _iRun:=400;
		ELSE
			 _iRun:=250;
		END_IF
	250:
		GVL.sErrorInfo:='';
		GVL.sErrorInfoTemp:="";
		GVL.sErrorInfoTemp:=WCONCAT(WCONCAT(WCONCAT(WCONCAT(WCONCAT(WCONCAT(WCONCAT(TO_WSTRING(_iErrorCode),","),TO_WSTRING( M_GetCategory(Category))),","),Language[Error.eSaveListLanguage]),","),SEL(Message="",Message,Language[E_Language.Chinese])),"$R");
		WSTRING_TO_UTF8(ADR(GVL.sErrorInfo),ADR(GVL.sErrorInfoTemp),SIZEOF(GVL.sErrorInfoTemp));
		_iRun:=300;
	300:
		GVL.FbErrorLog.AppendAllText:=TRUE;
		IF GVL.FbErrorLog.Done THEN
			GVL.FbErrorLog.AppendAllText:=FALSE;
			_iRun:=400;
		END_IF
	400:
		GVL.bFileErrorLogLock:=FALSE;
		_iRun:=500;
	500:
		IF NOT Error.bSaveErrorList THEN
			_iRun:=0;
		END_IF
END_CASE

END_FUNCTION_BLOCK

// Error/POUs/M_GetCategory
FUNCTION M_GetCategory : STRING
VAR_INPUT
	Category:				E_ErrorCategory;	
END_VAR
VAR
END_VAR

CASE Category OF
	E_ErrorCategory.Axis:
		M_GetCategory:= 'Axis';
	E_ErrorCategory.Cylinder:
		M_GetCategory:='Cylinder';
	E_ErrorCategory.Other:
		M_GetCategory:='Other';
	E_ErrorCategory.Safety:
		M_GetCategory:='Safety';
	E_ErrorCategory.Station:
		M_GetCategory:='Satation';
	E_ErrorCategory.TCP_IP:
		M_GetCategory:='TCP_IP';
END_CASE

END_FUNCTION

// System/POUs/FB_MemoryLag
FUNCTION_BLOCK FB_MemoryLag
VAR_INPUT
	Value:				LREAL;// 需要记忆的值
	Lag:				REAL;// 允许误差值
	ID:					BYTE;
	Category:			E_ErrorCategory;
	InfoIndex:			BYTE;
	System:				REFERENCE TO ST_System;
	Error:				REFERENCE TO ST_Error;
	Message:			WSTRING;// 提示信息
	Position:			WSTRING;// 实例位置
	Language:			ARRAY[0..E_Language.MaxCount] OF WSTRING;
END_VAR
VAR_OUTPUT
	Erroring:			BOOL;
	MemoryValue:		LREAL;
END_VAR
VAR
	_iRun:					INT;
	_fbErrorTag:			FB_ErrorTag;
	_ton:					TON;
	_log:					REAL;
	_i:						INT;
END_VAR

_ton(IN:=System.stMode.bAuto AND System.stMode.bStop , PT:= T#1S, Q=> , ET=> );
IF NOT _ton.Q  THEN
	MemoryValue:=Value;
END_IF

_log:=ABS(Lag);

_fbErrorTag(
	Error:=Error , 
	System:=System , 
	Enable:= , 
	Message:=, 
	Level:=5 , 
	Position:=Position , 
	ErrorTime:= ,
	Language:= ,
	Erroring=>Erroring,
	ID:=ID,
	Category:=Category,
	InfoIndex:=InfoIndex );
	
CASE _iRun OF
	0:
		_fbErrorTag.Enable:=FALSE;
		IF ABS(Value-MemoryValue)>_log THEN
			_iRun:=50;
		END_IF
	50:
		FOR _i:=0 TO E_Language.MaxCount BY 1 DO
			_fbErrorTag.Language[_i]:=WCONCAT(WCONCAT(Language[_i]," "), LREAL_TO_WSTRING(MemoryValue));
		END_FOR 
		_iRun:=100;
	100:
		_fbErrorTag.Enable:=TRUE;
		System.stMode.iMemory:=System.stMode.iMemory+1;
		_iRun:=200;
	200:
		IF ABS(Value-MemoryValue)<=_log THEN
			_iRun:=300;
		END_IF
	300:
		System.stMode.iMemory:=System.stMode.iMemory-1;
		_iRun:=0;
END_CASE

END_FUNCTION_BLOCK

// AxisCam/FB_AxisCam
FUNCTION_BLOCK FB_AxisCam
VAR_INPUT
	Execute:				BOOL;// 为真则耦合 为假则解偶
	Master:					REFERENCE TO ST_Axis;// 主轴
	Slave:					REFERENCE TO ST_Axis;// 从轴
	StartMode:				MC_StartMode:=MC_STARTMODE_ABSOLUTE;// 开始模式 默认为绝对定位
	CamTableID:				MC_CAM_ID:=100;// 凸轮ID
	ArrayTable:				POINTER TO MC_MotionFunctionPoint;//Arry(0..x) OF MC_MotionFunctionPoint
	ArrayCount:				UINT;// ArrayTable数量 从1开始
	ArraySize:				UDINT;// sizeof(MotionFunctionPoint)
END_VAR
VAR_OUTPUT
	Busy:					BOOL;
	Error:					BOOL;
	InSync:					BOOL;
	ErrorID:				UDINT;
END_VAR
VAR
	_mcCamIn:					MC_CamIn;
	_mcCamOut:					MC_CamOut;
	_mcCamTableSelect:			MC_CamTableSelect;
	_camTable:					MC_CAM_REF;
	_iRun:						UDINT;
END_VAR

_camTable.ArraySize:=ArraySize;
_camTable.NoOfColumns:=1;// 和TableType为固定值
_camTable.NoOfRows:=ArrayCount;
_camTable.pArray:=ArrayTable;
_camTable.TableType:=MC_TABLETYPE_MOTIONFUNCTION;// 函数在运行时计算

_mcCamTableSelect(
	Master:=Master.Axis_REF , 
	Slave:=Slave.Axis_REF, 
	CamTable:=_camTable , 
	Execute:= , 
	Periodic:= , 
	MasterAbsolute:= , 
	SlaveAbsolute:= , 
	CamTableID:=CamTableID , 
	Done=> , 
	Busy=> , 
	Error=> , 
	ErrorID=> );
	
_mcCamIn(
	Master:=Master.Axis_REF , 
	Slave:=Slave.Axis_REF, 
	Execute:= , 
	MasterOffset:= , 
	SlaveOffset:= , 
	MasterScaling:= , 
	SlaveScaling:= , 
	StartMode:= StartMode ,
	CamTableID:=CamTableID , 
	BufferMode:= , 
	Options:= , 
	InSync=>InSync , 
	Busy=> , 
	Active=> , 
	CommandAborted=> , 
	Error=> , 
	ErrorID=> );
	
_mcCamOut(
	Slave:= Slave.Axis_REF, 
	Execute:= , 
	Options:= , 
	Done=> , 
	Busy=> , 
	Error=> , 
	ErrorID=> );
	
IF _mcCamTableSelect.Error OR _mcCamIn.Error OR _mcCamOut.Error OR Master.stStatus.bError OR Slave.stStatus.bError THEN
	Error:=TRUE;
END_IF

IF _mcCamTableSelect.Error THEN
	ErrorID:=_mcCamTableSelect.ErrorID;
END_IF

IF _mcCamIn.Error THEN
	ErrorID:=_mcCamIn.ErrorID;
END_IF

IF _mcCamOut.Error THEN
	ErrorID:=_mcCamOut.ErrorID;
END_IF


A_Run();

ACTION A_Run:
{attribute'hide'}

CASE _iRun OF
	0:
		Busy:=FALSE;
		IF Execute THEN
			_iRun:=100;
		END_IF;
	100:
		Error:=FALSE;
		Busy:=TRUE;
		_mcCamTableSelect.Execute:=TRUE;
		IF _mcCamTableSelect.Done THEN
			_mcCamTableSelect.Execute:=FALSE;
			_iRun:=200;
		END_IF
		IF _mcCamTableSelect.Error THEN
			_mcCamTableSelect.Execute:=FALSE;
			_iRun:=10000;
		END_IF
	200:
		_mcCamIn.Execute:=TRUE;
		IF _mcCamIn.Error OR NOT Execute THEN
			_mcCamIn.Execute:=FALSE;
			_iRun:=10000;
		END_IF
	10000:
		_mcCamOut.Execute:=TRUE;
		IF _mcCamOut.Busy OR _mcCamOut.Done OR _mcCamOut.Error THEN
			_mcCamOut.Execute:=FALSE;
			_iRun:=11000;
		END_IF
	11000:
		IF NOT Execute THEN
			_iRun:=0;
		END_IF
END_CASE
END_ACTION

{attribute'hide'}
METHOD M_Semicircle : POINTER TO MC_MotionFunctionPoint// 半圆 ArrayCount 数据尽量为2的整数倍 MC_StartMode:=MC_STARTMODE_ABSOLUTE
VAR_INPUT
	Radius:							LREAL;// 半径
	A:								LREAL;// 圆心X
	B:								LREAL;// 圆心Y
END_VAR
VAR
	_temp:							LREAL;
	_i:								UINT;
	_temp1:							UINT;;
END_VAR
IF ArrayCount=0 THEN RETURN; END_IF
	
_temp:=2*Radius/ArrayCount;
_temp1:=DINT_TO_UINT(TRUNC(ArrayCount/2));

_i:=0;
ArrayTable[_i].FunctionType:=MOTIONFUNCTYPE_SPLINE;
ArrayTable[_i].MasterPos:=A-Radius;
ArrayTable[_i].SlavePos:=B;
ArrayTable[_i].PointIndex:=_i+1;
ArrayTable[_i].PointType:=MOTIONPOINTTYPE_MOTION;

_i:=ArrayCount-1;
ArrayTable[_i].FunctionType:=MOTIONFUNCTYPE_SPLINE;
ArrayTable[_i].MasterPos:=A+Radius;
ArrayTable[_i].SlavePos:=B;
ArrayTable[_i].PointIndex:=_i+1;
ArrayTable[_i].PointType:=MOTIONPOINTTYPE_MOTION;

FOR _i:=1 TO _temp1-1 BY 1 DO
	ArrayTable[_i].FunctionType:=MOTIONFUNCTYPE_SPLINE;
	ArrayTable[_i].MasterPos:=a-Radius+_temp*_i;
	ArrayTable[_i].SlavePos:=b+SQRT(Radius*Radius-(ArrayTable[_i].MasterPos-a)*(ArrayTable[_i].MasterPos-a));
	ArrayTable[_i].PointIndex:=_i+1;
	ArrayTable[_i].PointType:=MOTIONPOINTTYPE_MOTION;
END_FOR

FOR _i:=_temp1 TO ArrayCount-2 BY 1 DO
	ArrayTable[_i].FunctionType:=MOTIONFUNCTYPE_SPLINE;
	ArrayTable[_i].MasterPos:=a+_temp*(_i-_temp1);
	ArrayTable[_i].SlavePos:=b+SQRT(Radius*Radius-(ArrayTable[_i].MasterPos-a)*(ArrayTable[_i].MasterPos-a));
	ArrayTable[_i].PointIndex:=_i+1;
	ArrayTable[_i].PointType:=MOTIONPOINTTYPE_MOTION;
END_FOR

M_Semicircle:=ArrayTable;
END_METHOD

END_FUNCTION_BLOCK

// Convert/Data_TO_Data
FUNCTION Data_TO_Data
VAR_INPUT
	In:				POINTER TO BYTE;
	SizeIn:			UINT;
	Q:				POINTER TO BYTE;
	SizeQ:			UINT;
END_VAR
VAR
	_i:				UINT;
END_VAR

FOR _i:=0 TO SizeQ-1 BY 1 DO
	Q[_i]:=0;
END_FOR;

FOR _i:=0 TO SizeIn-1 BY 1 DO
	IF _i<=SizeQ-1 THEN
		Q[_i]:=In[_i];
	END_IF;
END_FOR;

END_FUNCTION

// CycleTime/FB_CycleTime
FUNCTION_BLOCK FB_CycleTime
VAR_INPUT
	Execute:				BOOL;
	System:					ST_System;
END_VAR
VAR_OUTPUT
	Busy:					BOOL;
	CycleTime:				TIME;// 由两次触发时间间隔得出
END_VAR
VAR
	_iRun:					UINT;
	_arrTon:				ARRAY[0..2] OF TON;
	_cycleTime:				TIME;
	_fTRIG:					F_TRIG;
END_VAR

_fTRIG(CLK:=NOT System.stMode.bStop AND Busy , Q=> );
IF _fTRIG.Q THEN
	_cycleTime:=_cycleTime+_arrTon[0].ET;
END_IF
_arrTon[0](IN:=_fTRIG.CLK , PT:=T#1100H , Q=> , ET=> );

IF System.stInput.bReset THEN
	_iRun:=0;
END_IF



CASE _iRun OF
	0:
		_cycleTime:=T#0S;
		_arrTon[0].IN:=Busy:=FALSE;
		IF Execute AND System.stMode.bAutoRunning THEN
			_iRun:=100;
		END_IF; 
	100:
		_arrTon[0].IN:=Busy:=TRUE;
		IF NOT Execute THEN
			_iRun:=200;
		END_IF
	200:
		IF Execute THEN
			CycleTime:=_cycleTime;
			Busy:=FALSE;
			_iRun:=300;
		END_IF
	300:
		
		IF NOT Execute THEN
			_iRun:=0;
		END_IF
END_CASE

END_FUNCTION_BLOCK

// CycleTime/FB_CycleTime1
FUNCTION_BLOCK FB_CycleTime1
VAR_INPUT
	Execute:			BOOL;
END_VAR
VAR_OUTPUT
	CycleTime:			TIME;
END_VAR
VAR
	_rTRIG:				R_TRIG;
	_fTRIG:				F_TRIG;
	_arrTon:			ARRAY[0..2] OF TON;
END_VAR

_rTRIG(CLK:= Execute, Q=> );

IF _rTRIG.Q THEN
	IF _arrTon[0].IN THEN
		CycleTime:=_arrTon[0].ET;	
	END_IF
	IF _arrTon[1].IN THEN
		CycleTime:=_arrTon[1].ET;
	END_IF
	IF _arrTon[0].IN THEN
		_arrTon[0].IN:=FALSE;
		_arrTon[1].IN:=TRUE;
	ELSE
		_arrTon[0].IN:=TRUE;
		_arrTon[1].IN:=FALSE;
	END_IF
END_IF

_arrTon[0](IN:= , PT:=T#1100H , Q=> , ET=> );
_arrTon[1](IN:= , PT:=T#1100H , Q=> , ET=> );

END_FUNCTION_BLOCK

// Cylinder/POUs/FB_Cylinder
FUNCTION_BLOCK FB_Cylinder
VAR_INPUT
	System:						REFERENCE TO ST_System;// 系统集合
	Cylinder:					REFERENCE TO ST_Cylinder;//  气缸控制集合
	Data:						REFERENCE TO ST_CylinderData;// 气缸数据集合
	Error:						REFERENCE TO ST_Error;// 错误集合
END_VAR
VAR_OUTPUT
END_VAR
VAR
	_tonHome:					TON;
	_tonWork:					TON;
	_arrFbError:				ARRAY [0..10] OF FB_ErrorTag;
	_rTRIG:						R_TRIG;
	_arrFbMemory:				ARRAY [0..2] OF FB_Memory;
	_bFirstCycle:				BOOL:=TRUE;
	_i:							INT;
	
	_arrTon:					ARRAY[0..10] OF TON;
END_VAR

Cylinder.sName:=Cylinder.arrInfo[System.stMode.eLanguage].sName;


IF Cylinder.stLock.bShield THEN
	RETURN;
END_IF


IF _bFirstCycle THEN
	A_Init();
END_IF



A_ControlRest();

A_Home();

A_Work();

A_Off();

A_Memory();

A_Error();

_bFirstCycle:=FALSE;

ACTION A_ControlRest:
{attribute'hide'}

IF System.stMode.stDeviceRest.bAuto THEN
	Cylinder.stControl.stHomeRequest.bAuto:=FALSE;
	Cylinder.stControl.stWorkRequest.bAuto:=FALSE;
	Cylinder.stControl.stOffRequest.bAuto:=FALSE;
END_IF;
IF System.stMode.stDeviceRest.bManual THEN
	Cylinder.stControl.stHomeRequest.bManual:=FALSE;
	Cylinder.stControl.stWorkRequest.bManual:=FALSE;
	Cylinder.stControl.stOffRequest.bManual:=FALSE;
END_IF;
END_ACTION

ACTION A_Error:
{attribute'hide'}

_arrFbError[0](
	Error:=Error , 
	System:=System , 
	Enable:=Cylinder.stOutput.bHome AND NOT Cylinder.stInput.bHome, 
	Message:=, 
	Level:=3 , 
	ErrorTime:=UDINT_TO_TIME(Data.iAlarmTime),
	Position:=WCONCAT("FB_Cylinder:",Cylinder.arrInfo[System.stMode.eLanguage].sName),
	Erroring=>Cylinder.stStatus.bErrorHome,
	ID:=Cylinder.ID,
	Category:=E_ErrorCategory.Cylinder,
	InfoIndex:=0);

_arrFbError[1](
	Error:=Error , 
	System:=System , 
	Enable:=Cylinder.stOutput.bWork AND NOT Cylinder.stInput.bWork, 
	Message:=,
	Level:=3 , 
	ErrorTime:= UDINT_TO_TIME(Data.iAlarmTime),
	Position:=WCONCAT("FB_Cylinder:",Cylinder.arrInfo[System.stMode.eLanguage].sName),
	Erroring=>Cylinder.stStatus.bErrorWork,
	ID:=Cylinder.ID,
	Category:=E_ErrorCategory.Cylinder,
	InfoIndex:=1 );	

_arrFbError[2](
	Error:=Error , 
	System:=System , 
	Enable:=Cylinder.stInput.bWork AND Cylinder.stInput.bHome, 
	Message:=, 
	Level:=3 , 
	ErrorTime:=UDINT_TO_TIME( Data.iAlarmTime),
	Position:=WCONCAT("FB_Cylinder:",Cylinder.arrInfo[System.stMode.eLanguage].sName),
	Erroring=>Cylinder.stStatus.bErrorTogether,
	ID:=Cylinder.ID,
	Category:=E_ErrorCategory.Cylinder,
	InfoIndex:=2);
END_ACTION

ACTION A_Home:
{attribute'hide'}
_arrTon[0](IN:=(System.stMode.stDeviceEnable.bAuto AND Cylinder.stControl.stHomeRequest.bAuto) , PT:=TO_TIME(Data.iHomeRequestTime) , Q=> , ET=> );

// 初始位
IF(_arrTOn[0].Q  OR (System.stMode.stDeviceEnable.bManual AND Cylinder.stControl.stHomeRequest.bManual)) AND NOT Cylinder.stLock.bHome AND NOT Cylinder.stLock.bAll THEN
	Cylinder.stOutput.bHome:=TRUE;
	Cylinder.stOutput.bWork:=FALSE;
END_IF;

_arrTon[1](IN:=Cylinder.stInput.bHome , PT:=TO_TIME(Data.iHomeDone) , Q=>Cylinder.stStatus.bHomeDone , ET=> );
END_ACTION

ACTION A_Init:
{attribute'hide'}

Cylinder.arrInfo[E_Language.Chinese].sHomeError:=":至初始位超时";
Cylinder.arrInfo[E_Language.Chinese].sWorkError:=":至工作位超时";
Cylinder.arrInfo[E_Language.Chinese].sWorkHomeError:=":初始位工作位传感器同时有信号";
Cylinder.arrInfo[E_Language.Chinese].sMemoryHome:=":初始位状态和记忆不符合";
Cylinder.arrInfo[E_Language.Chinese].sMemoryWork:=":工作位状态和记忆不符合";

Cylinder.arrInfo[E_Language.English].sHomeError:=": timeout to initial bit";
Cylinder.arrInfo[E_Language.English].sWorkError:=": timeout to workstation";
Cylinder.arrInfo[E_Language.English].sWorkHomeError:=": initial position working position sensor has signal simultaneously";
Cylinder.arrInfo[E_Language.English].sMemoryHome:=": Initial bit state and memory do not match";
Cylinder.arrInfo[E_Language.English].sMemoryWork:=": Work position state and memory do not match";

Cylinder.arrInfo[E_Language.Vietnamese].sHomeError:=": thời gian lên bit ban đầu";
Cylinder.arrInfo[E_Language.Vietnamese].sWorkError:=": đồng hồ làm việc";
Cylinder.arrInfo[E_Language.Vietnamese].sWorkHomeError:="Bộ cảm biến vị trí ban đầu có tín hiệu đồng thời";
Cylinder.arrInfo[E_Language.Vietnamese].sMemoryHome:="Trạng thái vị trí ban đầu và bộ nhớ không phù hợp";
Cylinder.arrInfo[E_Language.Vietnamese].sMemoryWork:="Trạng thái vị trí và trí nhớ không phù hợp";

Cylinder.arrInfo[E_Language.Hindi].sHomeError:=":प्रारंभिक बिट मध्यांतर के लिए";
Cylinder.arrInfo[E_Language.Hindi].sWorkError:=":समय से काम करने के लिए";
Cylinder.arrInfo[E_Language.Hindi].sWorkHomeError:=": काम करने की स्थिति सेंसर के प्रारंभिक बिट एक ही समय में एक संकेत है";
Cylinder.arrInfo[E_Language.Hindi].sMemoryHome:=": प्रारंभिक बिट राज्य और स्मृति मेल नहीं खाती";
Cylinder.arrInfo[E_Language.Hindi].sMemoryWork:=": काम करने की स्थिति राज्य और स्मृति के अनुरूप नहीं है";

FOR _i:=0 TO E_Language.MaxCount BY 1 DO
	_arrFbError[0].Language[_i]:=WCONCAT(Cylinder.arrInfo[_i].sName,Cylinder.arrInfo[_i].sHomeError);
	_arrFbError[1].Language[_i]:=WCONCAT(Cylinder.arrInfo[_i].sName,Cylinder.arrInfo[_i].sWorkError);
	_arrFbError[2].Language[_i]:=WCONCAT(Cylinder.arrInfo[_i].sName,Cylinder.arrInfo[_i].sWorkHomeError);
	
	_arrFbMemory[0].Language[_i]:=Cylinder.arrInfo[_i].sMemoryHome;
	_arrFbMemory[1].Language[_i]:=Cylinder.arrInfo[_i].sMemoryWork;
END_FOR;
END_ACTION

ACTION A_Memory:
{attribute'hide'}

_arrFbMemory[0](
	Value:=BOOL_TO_STRING(Cylinder.stOutput.bHome) , 
	System:=System , 
	Error:=Error , 
	Message:= , 
	Position:=WCONCAT("FB_Cylinder:",Cylinder.arrInfo[System.stMode.eLanguage].sName) , 
	Erroring=>Cylinder.stStatus.bMemoryHome,
	ID:=Cylinder.ID,
	Category:=E_ErrorCategory.Cylinder,
	InfoIndex:=20 );

	
_arrFbMemory[1](
	Value:=BOOL_TO_STRING(Cylinder.stOutput.bWork) , 
	System:=System , 
	Error:=Error , 
	Message:=, 
	Position:=WCONCAT("FB_Cylinder:",Cylinder.arrInfo[System.stMode.eLanguage].sName) , 
	Erroring=>Cylinder.stStatus.bMemoryWork,
	ID:=Cylinder.ID,
	Category:=E_ErrorCategory.Cylinder,
	InfoIndex:=21 );
END_ACTION

ACTION A_Off:
{attribute'hide'}
_arrTon[2](IN:=(System.stMode.stDeviceEnable.bAuto AND Cylinder.stControl.stOffRequest.bAuto ) , PT:=TO_TIME(Data.iOffRequestTime) , Q=> , ET=> );
// 释放请求
IF(_arrTon[2].Q  OR (System.stMode.stDeviceEnable.bManual AND Cylinder.stControl.stOffRequest.bManual)) AND NOT Cylinder.stLock.bOff AND NOT Cylinder.stLock.bAll THEN
	Cylinder.stOutput.bHome:=FALSE;
	Cylinder.stOutput.bWork:=FALSE;
END_IF;

_arrTon[3](IN:=NOT Cylinder.stOutput.bHome AND NOT Cylinder.stOutput.bWork , PT:=TO_TIME(Data.iOffDone) , Q=>Cylinder.stStatus.bOffDone , ET=> );
END_ACTION

ACTION A_Work:
{attribute'hide'}
_arrTon[4](IN:=System.stMode.stDeviceEnable.bAuto  AND Cylinder.stControl.stWorkRequest.bAuto , PT:=TO_TIME(Data.iWorkRequestTime) , Q=> , ET=> );
// 工作位
IF(_arrTon[4].Q OR (System.stMode.stDeviceEnable.bManual AND Cylinder.stControl.stWorkRequest.bManual)) AND NOT Cylinder.stLock.bWork AND NOT Cylinder.stLock.bAll THEN
	Cylinder.stOutput.bHome:=FALSE;
	Cylinder.stOutput.bWork:=TRUE;
END_IF;

_arrTon[5](IN:=Cylinder.stInput.bWork , PT:=TO_TIME(Data.iWorkDone) , Q=>Cylinder.stStatus.bWorkDone , ET=> );
END_ACTION

METHOD M_HomeRequest : BOOL
VAR_INPUT
END_VAR
Cylinder.stControl.stHomeRequest.bAuto:=TRUE;
Cylinder.stControl.stWorkRequest.bAuto:=FALSE;
Cylinder.stControl.stOffRequest.bAuto:=FALSE;

M_HomeRequest:=Cylinder.stStatus.bHomeDone;
END_METHOD

METHOD M_OffRequest : BOOL
VAR_INPUT
END_VAR
Cylinder.stControl.stOffRequest.bAuto:=TRUE;
Cylinder.stControl.stWorkRequest.bAuto:=FALSE;
Cylinder.stControl.stHomeRequest.bAuto:=FALSE;


M_OffRequest:=Cylinder.stStatus.bOffDone;
END_METHOD

METHOD M_WorkRequest : BOOL
VAR_INPUT
END_VAR
Cylinder.stControl.stHomeRequest.bAuto:=FALSE;
Cylinder.stControl.stWorkRequest.bAuto:=TRUE;
Cylinder.stControl.stOffRequest.bAuto:=FALSE;

M_WorkRequest:=Cylinder.stStatus.bWorkDone;
END_METHOD

END_FUNCTION_BLOCK

// System/POUs/FB_Memory
FUNCTION_BLOCK FB_Memory
VAR_INPUT
	ID:					BYTE;
	Category:			E_ErrorCategory;
	InfoIndex:			BYTE;
	Value:				STRING;// 需要记忆的值
	System:				REFERENCE TO ST_System;
	Error:				REFERENCE TO ST_Error;
	Message:			WSTRING;// 提示信息(中文)
	Position:			WSTRING;// 实例位置
	Language:			ARRAY[0..E_Language.MaxCount] OF WSTRING;
END_VAR
VAR_OUTPUT
	Erroring:			BOOL;
	MemoryValue:		STRING;
END_VAR
VAR
	_iRun:				INT;
	_fbErrorTag:		FB_ErrorTag;
	_ton:				TON;
	_i:					INT;
END_VAR

_ton(IN:=System.stMode.bAuto AND System.stMode.bStop , PT:= T#1S, Q=> , ET=> );
IF NOT _ton.Q  THEN
	MemoryValue:=Value;
END_IF;

_fbErrorTag(
	Error:=Error , 
	System:=System , 
	Enable:= , 
	Message:= , 
	Level:=5 , 
	Position:=Position , 
	ErrorTime:= ,
	Language:=, 
	Erroring=>Erroring,
	ID:=ID,
	Category:=Category,
	InfoIndex:=InfoIndex );


CASE _iRun OF
	0:
		_fbErrorTag.Enable:=FALSE;
		IF MemoryValue<>Value AND _ton.Q THEN
			_iRun:=50;
		END_IF;
	50:
		FOR _i:=0 TO E_Language.MaxCount BY 1 DO
			_fbErrorTag.Language[_i]:=WCONCAT(WCONCAT(Language[_i]," "),TO_WSTRING(MemoryValue));
		END_FOR 
		_iRun:=100;
	100:
		_fbErrorTag.Enable:=TRUE;
		System.stMode.iMemory:=System.stMode.iMemory+1;
		_iRun:=200;
	200:
		IF MemoryValue=Value THEN
			_iRun:=300;
		END_IF;
	300:
		System.stMode.iMemory:=System.stMode.iMemory-1;
		_iRun:=0;
END_CASE;

END_FUNCTION_BLOCK

// Error/POUs/FB_ErrorTagStation
FUNCTION_BLOCK FB_ErrorTagStation
VAR_INPUT
	StationIndex:			INT;// 工站索引
	Error:					REFERENCE TO ST_Error;
	System:					REFERENCE TO ST_System;
	ID:						BYTE;// ID(生成ErrorCode使用 如无相关需求可忽略)
	Category:				E_ErrorCategory;// 报警类别(生成ErrorCode使用 如无相关需求可忽略)
	InfoIndex:				BYTE;// 从50开始(生成ErrorCode使用 如无相关需求可忽略)
	Enable:					BOOL;// 报警触发
	Message:				WSTRING;// 报警内容
	Position:				WSTRING;// 错误发生位置
	ErrorTime:				TIME:=T#0S;// 报警延迟
	Language:				ARRAY[0..E_Language.MaxCount] OF WSTRING;//	其他语言集合
END_VAR
VAR_OUTPUT
	Erroring:				BOOL;// 通常用于触发第三方触摸屏(没有第三方屏幕时 此项可以不用填写)
	ErrorCode:				DWORD;
END_VAR
VAR
	_i:						INT;
	_iCyclic:				INT;
	_iRunNow:				INT;
	_tonError:				TON;
	_iTemp:					INT;
	_stNullInfo:			ST_ErrorInfo;
	_rTRIG:					R_TRIG;
	
	_iErrorCode:			DWORD;
	_pErrorCode:			POINTER TO BYTE;
	_arrErrorList:			ARRAY[0..10] OF STRING;
	_iRun:					UINT;
END_VAR

IF  _iCyclic<10 THEN
	_iCyclic:=_iCyclic+1;
	RETURN;
END_IF;

_tonError(IN:=Enable , PT:=ErrorTIME , Q=> , ET=> );

_pErrorCode:= ADR(_iErrorCode);
_pErrorCode[3]:=TO_BYTE(Category);
_pErrorCode[2]:=ID;
_pErrorCode[1]:=TO_BYTE(3);
_pErrorCode[0]:=InfoIndex;

IF System.stInput.bReset OR System.stInput.bResetAlarm  THEN
	Erroring:=FALSE;
	_iRunNow:=0;
END_IF;

// 记录当前报警
CASE _iRunNow OF
	0:
		_rTRIG.CLK:=FALSE;
		IF _tonError.Q AND NOT Erroring THEN
			_iRunNow:=100;
		END_IF;
	100:
		System.stMode.arrAlarmStation[StationIndex]:=TRUE;
		Erroring:=TRUE;
		_iRunNow:=200;
	200:
		_rTRIG.CLK:=TRUE;
		FOR _i:=0 TO Error.stNow.iCount BY 1 DO
			IF NOT Error.stNow.arrInfo[_i].bStatus THEN
				Error.stNow.arrInfo[_i].sSystemDate:=System.stSystemDate.sNow;
				Error.stNow.arrInfo[_i].bStatus:=TRUE;
				Error.stNow.arrInfo[_i].sLevel:=INT_TO_STRING(0);
				Error.stNow.arrInfo[_i].sPosition:=Position;
				Error.stNow.arrInfo[_i].arrMessage:=Language;
				Error.stNow.arrInfo[_i].iErrorCode:=_iErrorCode;
				IF Message<>"" THEN
					Error.stNow.arrInfo[_i].arrMessage[E_Language.Chinese]:=Message;
				END_IF;
				_iTemp:=_i;
				EXIT;
			END_IF;
		END_FOR;
		_iRunNow:=300;
	300:
		IF NOT Enable THEN
			_iRunNow:=0;
		END_IF;
END_CASE;

// 记录历史报警
_rTRIG(CLK:= , Q=> );
IF _rTRIG.Q THEN
	FOR _i:=Error.stHistory.iCount TO 1 BY -1 DO
		Error.stHistory.arrInfo[_i]:=Error.stHistory.arrInfo[_i-1];
	END_FOR;
	Error.stHistory.arrInfo[0].sSystemDate:=System.stSystemDate.sNow;
	Error.stHistory.arrInfo[0].arrMessage:=Language;
	Error.stHistory.arrInfo[0].sLevel:=INT_TO_STRING(0);
	Error.stHistory.arrInfo[0].sPosition:=Position;
	Error.stHistory.arrInfo[0].iErrorCode:=_iErrorCode;
	IF Message<>"" THEN
		Error.stHistory.arrInfo[0].arrMessage[E_Language.Chinese]:=Message;
	END_IF;
END_IF;

CASE _iRun OF
	0:
		IF Error.bSaveErrorList THEN
			_iRun:=100;
		END_IF
	100:
		IF NOT GVL.bFileErrorLogLock THEN
			GVL.bFileErrorLogLock:=TRUE;
			_iRun:=250;
		END_IF
	250:
		GVL.sErrorInfo:='';
		GVL.sErrorInfoTemp:="";
		GVL.sErrorInfoTemp:=WCONCAT(WCONCAT(WCONCAT(WCONCAT(WCONCAT(WCONCAT(WCONCAT(TO_WSTRING(_iErrorCode),","),TO_WSTRING( M_GetCategory(Category))),","),Language[Error.eSaveListLanguage]),","),SEL(Message="",Message,Language[E_Language.Chinese])),"$R");
		WSTRING_TO_UTF8(ADR(GVL.sErrorInfo),ADR(GVL.sErrorInfoTemp),SIZEOF(GVL.sErrorInfoTemp));
		_iRun:=300;
	300:
		GVL.FbErrorLog.AppendAllText:=TRUE;
		IF GVL.FbErrorLog.Done THEN
			GVL.FbErrorLog.AppendAllText:=FALSE;
			_iRun:=400;
		END_IF
	400:
		GVL.bFileErrorLogLock:=FALSE;
		_iRun:=500;
	500:
		IF NOT Error.bSaveErrorList THEN
			_iRun:=0;
		END_IF
END_CASE

END_FUNCTION_BLOCK

// File/POUs/FB_DirectoryHelper
FUNCTION_BLOCK FB_DirectoryHelper
VAR_INPUT
	Execute:						BOOL;
	Command:						E_Directory;
	DirectoryPath:					STRING;// 文件夹路径		
END_VAR
VAR_OUTPUT
	Busy:							BOOL;
	Error:							BOOL;
	Done:							BOOL;
END_VAR
VAR
	_fbCreateDir:					FB_CreateDir;
	_fbRemoveDir:					FB_RemoveDir;
	_iRun:							UINT;
END_VAR

_fbCreateDir(
	sNetId:= , 
	sPathName:=DirectoryPath , 
	ePath:= , 
	bExecute:= , 
	tTimeout:= , 
	bBusy=> , 
	bError=> , 
	nErrId=> );
	
_fbRemoveDir(
	sNetId:= , 
	sPathName:=DirectoryPath , 
	ePath:= , 
	bExecute:= , 
	tTimeout:= , 
	bBusy=> , 
	bError=> , 
	nErrId=> );

A_Run();

ACTION A_Run:
CASE _iRun OF
	0:
		Done:=Busy:=FALSE;
		_fbCreateDir.bExecute:=FALSE;
		_fbRemoveDir.bExecute:=FALSE;
		IF Execute THEN
			_iRun:=100;
		END_IF
	100:
		Busy:=TRUE;
		Error:=FALSE;
		CASE Command OF
			E_Directory.Create:
				_fbCreateDir.bExecute:=TRUE;
			E_Directory.Delete:
				_fbRemoveDir.bExecute:=TRUE;
			ELSE
				Error:=TRUE;
				_iRun:=10000;
		END_CASE
		_iRun:=200;
	200:
		IF _fbCreateDir.bBusy OR _fbRemoveDir.bBusy THEN
			_iRun:=300;
		END_IF
	300:
		IF NOT _fbCreateDir.bBusy AND NOT _fbRemoveDir.bBusy  THEN
			_iRun:=400;
		END_IF
	400:
		CASE Command OF
			E_Directory.Create:
				Error:=_fbCreateDir.bError;
			E_Directory.Delete:
				Error:=_fbRemoveDir.bError;
		END_CASE
		_iRun:=10000;
	10000:
		Busy:=FALSE;
		Done:=TRUE;
		IF NOT Execute THEN
			_iRun:=0;
		END_IF
END_CASE
END_ACTION

END_FUNCTION_BLOCK

// File/POUs/FB_DirectoryHelper1
FUNCTION_BLOCK FB_DirectoryHelper1
VAR_INPUT
	Execute:						BOOL;
	Command:						E_Directory;
	FolderPath:						STRING;// 文件夹路径		
END_VAR
VAR_OUTPUT
	Busy:							BOOL;
	Error:							BOOL;
	Done:							BOOL;
END_VAR
VAR
	_fbWindowsCmd:					FB_WindowsCmd;
	_cmdTemp:						STRING;
	_rTRIG:								R_TRIG;
END_VAR

_rTRIG(CLK:=Execute , Q=> );

IF _rTRIG.Q THEN
	CASE Command OF
		E_Directory.Create:
			_cmdTemp:=CONCAT('md ' ,FolderPath);
		E_Directory.Delete:
			_cmdTemp:=CONCAT('rd /s /q '  ,FolderPath);
	END_CASE
END_IF

_fbWindowsCmd(
	Execute:=Execute , 
	Command:=ADR(_cmdTemp),
	Busy=> , 
	Done=> , 
	Error=> );

END_FUNCTION_BLOCK

// Windows/FB_WindowsCmd
FUNCTION_BLOCK FB_WindowsCmd
VAR_INPUT
	Execute:				BOOL;// 触发使能(在收到Done后 才能False)
	Command:				PVOID;
END_VAR
VAR_OUTPUT
	Busy:					BOOL;
	Done:					BOOL;
	Error:					BOOL;
END_VAR
VAR
	_fbFielHelper:			FB_FileHelper;
	_StartProcess:			NT_StartProcess;	
	_run:					UINT;
	_path:					STRING;
	_ton:					TON;
END_VAR

_fbFielHelper.FilePath:=_StartProcess.PATHSTR:='C:\TwinCAT\WindowsCmdTemp.bat';
_ton(IN:= , PT:=T#0.5S , Q=> , ET=> );

_StartProcess(
	NETID:= , 
	PATHSTR:= , 
	DIRNAME:='C:\TwinCAT\' , 
	COMNDLINE:= , 
	START:= , 
	TMOUT:= , 
	BUSY=> , 
	ERR=> , 
	ERRID=> );
	
_fbFielHelper(
	Read:= , 
	WriteAllText:= , 
	AppendAllText:= , 
	FilePath:= , 
	Buffer:=Command , 
	BufferLen:=F_LEN(Command) , 
	TimeOut:= , 
	Busy=> , 
	Error=> , 
	Done=> );
	
A_Run();

ACTION A_Run:
{attribute'hide'}
IF (_fbFielHelper.Error OR _StartProcess.ERR) AND Done THEN
	Error:=TRUE;
END_IF;

CASE _run OF 
	0:
		_fbFielHelper.WriteAllText:=FALSE;
		_StartProcess.START:=FALSE;
		Busy:=Done:=FALSE;
		IF Execute THEN
			_run:=100;
		END_IF
	100:
		Busy:=TRUE;
		Error:=FALSE;
		IF NOT GVL.bWindowsCmdLock THEN
			GVL.bWindowsCmdLock:=TRUE;
			_run:=200;
		END_IF
	200:
		_fbFielHelper.WriteAllText:=TRUE;
		IF  _fbFielHelper.Done THEN
			_fbFielHelper.WriteAllText:=FALSE;
			_run:=SEL(_fbFielHelper.Error,300,1000);
		END_IF
	300:
		_StartProcess.START:=TRUE;
		IF _StartProcess.BUSY THEN
			_run:=400;
		END_IF
	400:
		_StartProcess.START:=FALSE;
		IF NOT _StartProcess.BUSY THEN
			_run:=1000;
		END_IF
	1000:
		_ton.IN:=TRUE;
		IF _ton.Q THEN
			_ton.IN:=GVL.bWindowsCmdLock:=FALSE;
			_run:=1100;
		END_IF
	1100:
		Busy:=FALSE;
		Done:=TRUE;
		IF NOT Execute THEN
			Done:=FALSE;
			_run:=0;
		END_IF;
END_CASE
END_ACTION

END_FUNCTION_BLOCK

// Regex/F_LEN
FUNCTION F_LEN : UDINT
VAR_INPUT
	In:						POINTER TO BYTE;
END_VAR
VAR
	_i:						UDINT;
END_VAR

F_LEN:=0;
WHILE In[F_LEN]<>0 DO
	F_LEN:=F_LEN+1;
END_WHILE

END_FUNCTION

// File/POUs/FB_FileHelper
FUNCTION_BLOCK FB_FileHelper
VAR_INPUT
	Read:					BOOL;
	WriteAllText:			BOOL;
	AppendAllText:			BOOL;
	FilePath:				STRING;
	Buffer:					PVOID;
	BufferLen:				UDINT;
	TimeOut:				TIME:=T#2S;
END_VAR
VAR_OUTPUT
	Busy:					BOOL;
	Error:					BOOL;
	Done:					BOOL;				
END_VAR
VAR
	_run:					UINT;
	_ton:					TON;
	FileOpen : 				Tc2_System.FB_FileOpen;
	FileRead : 				Tc2_System.FB_FileRead;
	FileWrite : 			Tc2_System.FB_FileWrite;
	FileClose : 			Tc2_System.FB_FileClose;
END_VAR

FileOpen(
		sPathName:= FilePath, 
		nMode:= ,
		ePath:= , 
		bExecute:=);
FileRead(
		hFile:= FileOpen.hFile, 
		pReadBuff:=Buffer, 
		cbReadLen:= BufferLen, 
		bExecute:= );
FileWrite(
		hFile:= FileOpen.hFile, 
		pWriteBuff:= Buffer, 
		cbWriteLen:= F_LEN(Buffer), 
		bExecute:=);
FileClose(
		hFile:= FileOpen.hFile, 
		bExecute:=);
			
IF (FileOpen.bError OR FileRead.bError OR FileWrite.bError OR FileClose.bError) AND Done THEN
	Error:=TRUE;
END_IF
_ton(IN:=, PT:=TimeOut , Q=> , ET=> );
IF _ton.Q THEN
	_run:=1000;
	Error:=TRUE;
END_IF
			
			
CASE _run OF
	0:
		_ton.IN:=Done:=Busy:=FALSE;
		FileOpen.bExecute := FALSE;
		FileRead.bExecute := FALSE;
		FileClose.bExecute := FALSE;
		IF Read OR WriteAllText OR AppendAllText THEN
			_ton.IN:=TRUE;
			_run:=100;
		END_IF;
	100:
		Error:=FALSE;
		IF Read THEN
			FileOpen.nMode:=FOPEN_MODEREAD;
		END_IF
		IF WriteAllText THEN
			FileOpen.nMode:=FOPEN_MODEWRITE OR FOPEN_MODEPLUS;
		END_IF
		IF AppendAllText THEN
			FileOpen.nMode:=FOPEN_MODEAPPEND;
		END_IF
		_run:=110;
	110:
		FileOpen.bExecute:=TRUE;
		IF FileOpen.bBusy THEN
			_run := 120;
		END_IF
	120:
		FileOpen.bExecute:=FALSE;
		IF NOT FileOpen.bBusy THEN
			_run :=SEL(FileOpen.bError,200,1000);
		END_IF
	200:
		Busy:=TRUE;
		IF Read THEN
			_run := 300;
		END_IF
		IF WriteAllText OR AppendAllText THEN
			_run := 400;
		END_IF
		IF NOT Read AND NOT WriteAllText AND NOT AppendAllText THEN
			_run:=0;
		END_IF
	300:
		FileRead.bExecute:=TRUE;
		IF FileRead.bBusy THEN
			_run:=310;
		END_IF
	310:
		FileRead.bExecute:=FALSE;
		IF NOT FileRead.bBusy THEN
			_run :=1000;
		END_IF
	400:
		FileWrite.bExecute:=TRUE;
		IF FileWrite.bBusy THEN
			_run:=410;
		END_IF
	410:
		FileWrite.bExecute:=FALSE;
		IF NOT FileWrite.bBusy THEN
			_run :=1000;
		END_IF
	1000:
		_ton.IN:=FALSE;
		FileClose.bExecute:=TRUE;
		IF FileClose.bBusy THEN
			_run :=1100;
		END_IF
	1100:
		FileClose.bExecute:=FALSE;
		IF NOT FileClose.bBusy THEN
			_run :=1200;
		END_IF
	1200:
		Done:=TRUE;
		Busy:=FALSE;
		IF NOT Read AND NOT WriteAllText AND NOT AppendAllText  THEN
			Done:=FALSE;
			_run:=0;
		END_IF
END_CASE

END_FUNCTION_BLOCK

// File/POUs/FB_FileHandle
FUNCTION_BLOCK FB_FileHandle
VAR_INPUT
	FileHandle:				REFERENCE TO ST_FileHandle;
	Data:					REFERENCE TO ST_FileHandleData;
	System:					REFERENCE TO ST_System;
	Error:					REFERENCE TO ST_Error;
END_VAR
VAR
	_iRun:						INT;
	_bRead:						BOOL;
	_bWrite:					BOOL;
	_sWriteData:				STRING(255);
	_i:							INT;
	_t:							INT;
END_VAR
VAR
	_fbFileOpen:				FB_FileOpen;
	_fbFileGets:				FB_FileGets;
	_fbFileWrite:				FB_FileWrite;
	_fbFileClose:				FB_FileClose;
	_fbErrorTag:				ARRAY[0..3] OF FB_ErrorTag;
END_VAR

_fbFileOpen(
	sNetId:= , 
	sPathName:=Data.sFilePath , 
	nMode:= , 
	ePath:=PATH_GENERIC , 
	bExecute:= , 
	tTimeout:= , 
	bBusy=> , 
	bError=> , 
	nErrId=> , 
	hFile=> );
	
_fbFileGets(
	sNetId:= , 
	hFile:=_fbFileOpen.hFile , 
	bExecute:= , 
	tTimeout:= , 
	bBusy=> , 
	bError=> , 
	nErrId=> , 
	sLine=> , 
	bEOF=> );

_sWriteData:=CONCAT(FileHandle.sWriteBuffer,'$N');		
_fbFileWrite(
	sNetId:= , 
	hFile:=_fbFileOpen.hFile , 
	pWriteBuff:=ADR(_sWriteData) , 
	cbWriteLen:=LEN(_sWriteData) , 
	bExecute:= , 
	tTimeout:= , 
	bBusy=> , 
	bError=> , 
	nErrId=> , 
	cbWrite=> );
	
_fbFileClose(
	sNetId:= , 
	hFile:=_fbFileOpen.hFile , 
	bExecute:= , 
	tTimeout:= , 
	bBusy=> , 
	bError=> , 
	nErrId=> );
	
A_Error();

A_Read();

A_Rest();

A_Status();

A_Write();

A_Run();

ACTION A_Error:
{attribute'hide'}

_fbErrorTag[0](
	Error:=Error , 
	System:=System , 
	Enable:=_fbFileOpen.bError , 
	Message:=WCONCAT(FileHandle.sName,WCONCAT(":文件打开错误",UDINT_TO_WSTRING(_fbFileOpen.nErrId))) , 
	Level:=4 , 
	ErrorTime:=,
	Position:=WCONCAT("FB_FileHandle:",FileHandle.sName),
	Erroring=>FileHandle.stStatus.bErrorOpen,
	ID:=FileHandle.ID,
	Category:=E_ErrorCategory.File,
	InfoIndex:=0 );
	
_fbErrorTag[1](
	Error:=Error , 
	System:=System , 
	Enable:=_fbFileGets.bError , 
	Message:=WCONCAT(FileHandle.sName,WCONCAT(":文件读取错误",UDINT_TO_WSTRING(_fbFileGets.nErrId))) , 
	Level:=4 , 
	ErrorTime:=,
	Position:=WCONCAT("FB_FileHandle:",FileHandle.sName),
	Erroring=>FileHandle.stStatus.bErrorGet,
	ID:=FileHandle.ID,
	Category:=E_ErrorCategory.File,
	InfoIndex:=1 );
	
_fbErrorTag[2](
	Error:=Error , 
	System:=System , 
	Enable:=_fbFileWrite.bError , 
	Message:=WCONCAT(FileHandle.sName,WCONCAT(":文件写入错误",UDINT_TO_WSTRING(_fbFileWrite.nErrId))) , 
	Level:=4 , 
	ErrorTime:= ,
	Position:=WCONCAT("FB_FileHandle:",FileHandle.sName),
	Erroring=>FileHandle.stStatus.bErrorWrite,
	ID:=FileHandle.ID,
	Category:=E_ErrorCategory.File,
	InfoIndex:=2 );
	
_fbErrorTag[3](
	Error:=Error , 
	System:=System , 
	Enable:=_fbFileClose.bError , 
	Message:=WCONCAT(FileHandle.sName,WCONCAT(":文件关闭错误",UDINT_TO_WSTRING(_fbFileClose.nErrId))) , 
	Level:=4 , 
	ErrorTime:=,
	Position:=WCONCAT("FB_FileHandle:",FileHandle.sName),
	Erroring=>FileHandle.stStatus.bErrorClose,
	ID:=FileHandle.ID,
	Category:=E_ErrorCategory.File,
	InfoIndex:=3  );
END_ACTION

ACTION A_Read:
{attribute'hide'}

IF (System.stMode.stDeviceEnable.bManual AND FileHandle.stControl.stRead.bAuto) OR (System.stMode.stDeviceEnable.bManual AND FileHandle.stControl.stRead.bManual) THEN
	_bRead:=TRUE;
	_fbFileOpen.nMode:=FOPEN_MODEREAD;
ELSE
	_bRead:=FALSE;
END_IF
END_ACTION

ACTION A_Rest:
{attribute'hide'}

IF System.stMode.stDeviceRest.bAuto THEN
	FileHandle.stControl.stRead.bAuto:=FALSE;
	FileHandle.stControl.stWrite.bAuto:=FALSE;
END_IF

IF System.stMode.stDeviceRest.bManual THEN
	FileHandle.stControl.stRead.bManual:=FALSE;
	FileHandle.stControl.stWrite.bManual:=FALSE;
END_IF
END_ACTION

ACTION A_Run:
{attribute'hide'}

IF FileHandle.stStatus.bError OR (NOT _bRead AND NOT _bWrite) THEN
	_iRun:=0;
END_IF

CASE _iRun OF
	0:
		_i:=0;
		_fbFileOpen.bExecute:=FALSE;
		_fbFileClose.bExecute:=FALSE;
		_fbFileWrite.bExecute:=FALSE;
		_fbFileGets.bExecute:=FALSE;
		FileHandle.stStatus.bDone:=FALSE;
		IF _bRead OR _bWrite THEN
			_iRun:=100;
		END_IF
	100:
		_fbFileOpen.bExecute:=TRUE;
		IF _fbFileOpen.bBusy  THEN
			_iRun:=200;
		END_IF
	200:
		IF NOT _fbFileOpen.bBusy  THEN
			_fbFileOpen.bExecute:=FALSE;
			IF _bRead THEN
				_iRun:=205;
			END_IF
			IF _bWrite THEN
				_iRun:=300;
			END_IF
		END_IF
	205:
		FOR _t:=0 TO FileHandle.stReadBuffer.iCount BY 1DO
			FileHandle.stReadBuffer.arrBuffer[_t]:='';
		END_FOR
		_iRun:=210;
	210:
		_fbFileGets.bExecute:=TRUE;
		IF _fbFileGets.bBusy  THEN
			_iRun:=220;
		END_IF
	220:
		IF NOT _fbFileGets.bBusy THEN
			FileHandle.stReadBuffer.arrBuffer[_i]:=_fbFileGets.sLine;
			_fbFileGets.bExecute:=FALSE;
			_iRun:=230;
		END_IF
	230:
		IF _fbFileGets.bEOF OR _i>FileHandle.stReadBuffer.iCount THEN
			_iRun:=500;
		ELSE
			_i:=_i+1;
			_iRun:=210;
		END_IF
	300:
		_fbFileWrite.bExecute:=TRUE;
		IF _fbFileWrite.bBusy  THEN
			_iRun:=400;
		END_IF
	400:
		IF NOT _fbFileWrite.bBusy THEN
			_fbFileWrite.bExecute:=FALSE;
			_iRun:=500;
		END_IF
	500:
		_fbFileClose.bExecute:=TRUE;
		IF _fbFileClose.bBusy  THEN
			_iRun:=600;
		END_IF
	600:
		IF NOT _fbFileClose.bBusy THEN
			_fbFileClose.bExecute:=FALSE;
			_iRun:=700;
		END_IF
	700:
		FileHandle.stStatus.bDone:=TRUE;
		FileHandle.stReadBuffer.iLength:=_i;
		IF NOT  _bRead AND NOT  _bWrite  THEN
			_iRun:=0;
		END_IF
END_CASE
END_ACTION

ACTION A_Status:
{attribute'hide'}

FileHandle.stStatus.bBusy:= _fbFileOpen.bBusy OR _fbFileGets.bBusy OR _fbFileWrite.bBusy OR _fbFileClose.bBusy;

FileHandle.stStatus.bError:=_fbFileOpen.bError OR _fbFileGets.bError OR _fbFileWrite.bError OR _fbFileClose.bError;
END_ACTION

ACTION A_Write:
{attribute'hide'}

IF (System.stMode.stDeviceEnable.bAuto AND FileHandle.stControl.stWrite.bAuto) OR (System.stMode.stDeviceEnable.bManual AND FileHandle.stControl.stWrite.bManual) THEN
	_bWrite:=TRUE;
	_fbFileOpen.nMode:=FOPEN_MODEAPPEND;
ELSE
	_bWrite:=FALSE;
END_IF
END_ACTION

END_FUNCTION_BLOCK

// File/POUs/FB_LogHelper
FUNCTION_BLOCK FB_LogHelper // 不带缓存的Log文件写入
VAR_INPUT
	Execute:				BOOL;
	FilePath:				STRING;
	Message:				WSTRING(255);
END_VAR
VAR_OUTPUT
	Done:					BOOL;
	Busy:					BOOL;
	Error:					BOOL;
	ErrId:					INT;// 暂未使用
END_VAR
VAR
	_iRun:					INT;
	_fbFileOpen:			FB_FileOpen;
	_fbFileWrite:			FB_FileWrite;
	_fbFileClose:			FB_FileClose;
	_sTempString:			STRING(1000);
	_sTempWString:			WSTRING(1000);
END_VAR

_fbFileOpen(
	sNetId:= , 
	sPathName:=FilePath , 
	nMode:=FOPEN_MODEAPPEND , 
	ePath:= , 
	bExecute:= , 
	tTimeout:= , 
	bBusy=> , 
	bError=> , 
	nErrId=> , 
	hFile=> );
	
_sTempWString:=WCONCAT(Message,"$N");
WSTRING_TO_UTF8(ADR(_sTempString),ADR(_sTempWString),SIZEOF(_sTempWString));   
_fbFileWrite(
	sNetId:= , 
	hFile:=_fbFileOpen.hFile , 
	pWriteBuff:=ADR(_sTempString) , 
	cbWriteLen:=INT_TO_UDINT(LEN(_sTempString)) , 
	bExecute:= , 
	tTimeout:= , 
	bBusy=> , 
	bError=> , 
	nErrId=> , 
	cbWrite=> );

